	// Alarm_0403	403	Error	Wartość zadana wysokości jest większa od maksymalnej - zmień ustawienia w recepturze {0}
	//Error 7 - Bład nastaw max
	IF tonMaxHeightError.Q  THEN
		arfbAlarm[3].ipArguments.Clear() .AddLReal(lrMaxHeight);
		IF NOT arfbAlarm[3].bActive THEN
// 			bHeightMotorUp:=FALSE;
// 			bHeightMotorDown:=FALSE;
			arfbAlarm[3].Raise(nTimeStamp:=0);
		END_IF
	ELSE	
		IF  arfbAlarm[3].bActive AND bReset THEN
			arfbAlarm[3].Clear(nTimeStamp:=0, bResetConfirmation:= FALSE);
		END_IF	
// 		bError:=TRUE;
// 		udiErrorID:=7;
// 		udiErrorID:= udiErrorID+udiStationIndex;
// 		sErrorDescription:='Wartość zadana wysokości jest większa od maksymalnej - zmień ustawienia w recepturze';
// 		sErrorDescription2:=REAL_TO_STRING(LREAL_TO_INT(lrMaxHeight));
	END_IF
	// Alarm_0404	404	Error	Wartość zadana wysokości jest mniejsza od minimalnej - zmień ustawienia w recepturze {0}
	//Error 8 - Bład nastaw min
	IF tonMinHeightError.Q THEN
			arfbAlarm[4].ipArguments.Clear() .AddLReal(lrMinHeight);
		IF NOT arfbAlarm[4].bActive THEN
// 			bHeightMotorUp:=FALSE;
// 			bHeightMotorDown:=FALSE;
			arfbAlarm[4].Raise(nTimeStamp:=0);
		END_IF
	ELSE	
		IF  arfbAlarm[4].bActive AND bReset THEN
			arfbAlarm[4].Clear(nTimeStamp:=0, bResetConfirmation:= FALSE);
		END_IF
// 		bError:=TRUE;
// 		udiErrorID:=8;
// 		udiErrorID:= udiErrorID+udiStationIndex;
// 		sErrorDescription:='Wartość zadana wysokości jest mniejsza od minimalnej - zmień ustawienia w recepturze ';
// 		sErrorDescription2:=REAL_TO_STRING(LREAL_TO_INT(lrMinHeight));
	END_IF	
	// Alarm_0405	405	Error	Błąd falownika
	//Error 8 - Bład falownika
	IF tonInverterError.Q THEN
		IF NOT arfbAlarm[5].bActive THEN
			arfbAlarm[5].Raise(nTimeStamp:=0);
		END_IF
		IF arfbAlarm[5].bActive AND bReset THEN
			fbInverter.bReset := TRUE;
		END_IF
	ELSE	
		IF  arfbAlarm[5].bActive AND bReset THEN
			arfbAlarm[5].Clear(nTimeStamp:=0, bResetConfirmation:= FALSE);
		END_IF
// 		bError:=TRUE;
// 		udiErrorID:=9;
// 		udiErrorID:= udiErrorID+udiStationIndex;
// 		sErrorDescription:='Błąd falownika';
// 		sErrorDescription2:='';
	END_IF		
	
	
	
ELSE
	bError	:=FALSE;
END_IF


//-----------------------------------------------------------------------
IF bError AND NOT bStateError THEN

	IF eLastState = eRunning THEN
		bCycleNotDone						:= TRUE;
	END_IF

	eState 									:= E_Station.eError;
END_IF


//------------------------------------------------------------------------

(*Wyświetlanie błedu na wyjściu*)
bError							:= FALSE;
FOR nAlarmNumerator := 0 TO 19 DO
	bError						:= bError OR arfbAlarm[nAlarmNumerator].bActive;
END_FOR

(*Przepisywanie nazwy stacji*)
sErrorStationName 							:= WSTRING_TO_STRING(sStationName);

//Jezeli nie zbazowane to potrzebne bazowanie
IF NOT bHeightMotorEncoderHomed  THEN
	bHomingDone								:=	FALSE;
END_IF
END_ACTION

ACTION ACT_HeightMotor:
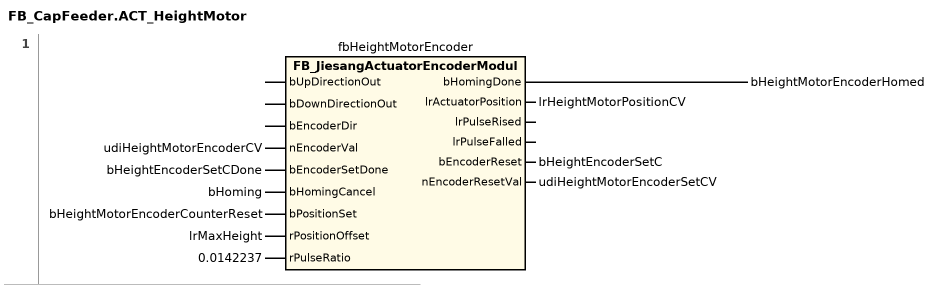
// NETWORK 1
fbHeightMotorEncoder(
    nEncoderVal := udiHeightMotorEncoderCV,
    bEncoderSetDone := bHeightEncoderSetCDone,
    bHomingCancel := bHoming,
    bPositionSet := bHeightMotorEncoderCounterReset,
    rPositionOffset := lrMaxHeight,
    rPulseRatio := 0.0142237,
    lrActuatorPosition => lrHeightMotorPositionCV,
    bEncoderReset => bHeightEncoderSetC,
    nEncoderResetVal => udiHeightMotorEncoderSetCV); // FB_JiesangActuatorEncoderModul
bHeightMotorEncoderHomed := fbHeightMotorEncoder.bHomingDone;
END_ACTION

ACTION ACT_Homing:
//BAZOWANIE

tofHeightMotorDown(IN:=bHeightMotorDown, PT:=T#1S); //Zabezpieczenie przed zbyt szybkim przełączeniem pomiędzy Down a Up, bezpiecznieki sie palą
	
//Podnoszenie stacji do maksymalnej pozycji
IF NOT bHeightMotorEncoderHomed OR rtEncoderHomed.Q THEN
	bHeightMotorUp:=(*TRUE*) NOT tofHeightMotorDown.Q AND NOT tonHomingSensor.Q;
	bHeightMotorDown:=FALSE;
	IF tonHeightNoChange.Q OR tonHeightNoChangeTime.Q THEN
		bHeightMotorEncoderCounterReset:=TRUE;
		bHeightMotorUp:=FALSE;
    END_IF
	//Jesli enkoder zbazowany zakończ bazowanie	
	IF rtEncoderHomed.Q  THEN
		bHeightMotorUp:=FALSE;
		bHeightMotorDown:=FALSE;
		eState:=E_Station.eHomingDone;
	END_IF		
		
//Po podniesieniu stacji opuszczanie do ustalonej wysokości
ELSIF bHeightMotorEncoderHomed THEN
	bHeightMotorEncoderCounterReset:=FALSE;
	bHeightMotorUp:=lrHeightMotorPositionCV<=lrHeightMotorPositionSV;
	bHeightMotorDown:=lrHeightMotorPositionCV>=lrHeightMotorPositionSV;
	//Kiedy stacja osiągnie wysokość zadaną
	IF ABS(lrHeightMotorPositionCV-lrHeightMotorPositionSV)<0.5 OR tonLimitPosMaxReachedDelay.Q OR tonLimitPosMinReachedDelay.Q THEN
		bHeightMotorDown:=FALSE;
		bHeightMotorUp:=FALSE;
		eState:=E_Station.eHomingDone;
	END_IF			
END_IF
END_ACTION

ACTION ACT_Inverter:
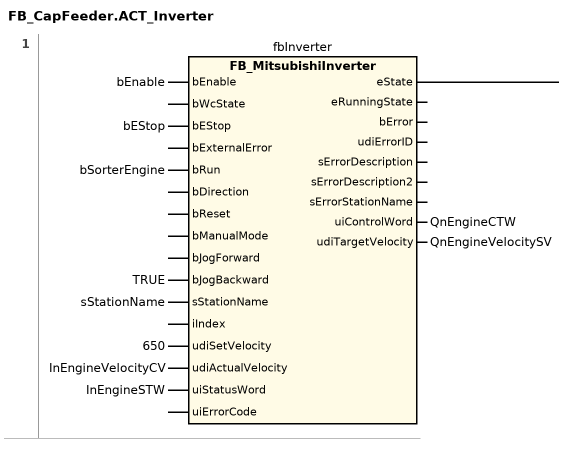
// NETWORK 1
fbInverter(
    bEnable := bEnable,
    bEStop := bEStop,
    bRun := bSorterEngine,
    bJogBackward := TRUE,
    sStationName := sStationName,
    udiSetVelocity := 650,
    udiActualVelocity := InEngineVelocityCV,
    uiStatusWord := InEngineSTW,
    uiControlWord => QnEngineCTW,
    udiTargetVelocity => QnEngineVelocitySV); // FB_MitsubishiInverter
END_ACTION

ACTION ACT_Limits:
IF iTimeToEmptySleeveError < 5 THEN
	iTimeToEmptySleeveError := 5;
END_IF
END_ACTION

ACTION ACT_ManualMovements:
//W trybie ruchów manualnych wykonuj ruchy za pomocą rozkazów manualnych
IF NOT bRun THEN
	
	bHeightMotorUp:=bManualHeightMotorUp;
	bHeightMotorDown:=bManualHeightMotorDown;
	bSorterEngine:=bManualSorterEngine;
	bSorterAir:=bManualSorterAir;
	
	bGate1:=bManualGate1; //Not dla tego, że defoltowy stan WYSUNIĘTY (true)
	bGate2:=bManualGate2; //Not dla tego, że defoltowy stan WYSUNIĘTY (true)

(*ELSE	//Kasuje zeby po cyklu nic sie nie poruszało

	bManualHeightMotorUp 	:= FALSE;
	bManualHeightMotorDown  := FALSE;
	bSorterEngine	:=FALSE;
	bSorterAir		:=FALSE;
*)	
END_IF


IF bHoming OR bHeightSet THEN
	eState:=E_Station.eHoming;
END_IF

IF bRun THEN	
	ACT_Running();
END_IF
//Zabezpieczenie przed kolizją stacji poprzez ruch podnośnika	
IF bHeightMotorDown AND lrHeightMotorPositionCV<=lrMinHeight AND NOT bHoming AND NOT bHeightSet THEN
	bHeightMotorDown:=FALSE;
END_IF	

IF bHeightMotorUp AND lrHeightMotorPositionCV>=lrMaxHeight AND NOT bHoming AND NOT bHeightSet THEN
	bHeightMotorUp:=FALSE;
END_IF
END_ACTION

ACTION ACT_ResetCommands:
//Reset komend ruchu 	


bHeightMotorUp				:=	FALSE;
bHeightMotorDown			:=	FALSE;
bSorterAir 		:= 	FALSE;
bSorterEngine 		:=	FALSE;
END_ACTION

ACTION ACT_Running:
//----------------------------------------------------------------------------------
// Obsługa podajnik zamknięc


(*CASE iValvesCycleCase OF
	0:
		bGate1:= FALSE;
		IF (tonGates1.Q) THEN
			iValvesCycleCase :=1;
		END_IF
	1:
		bGate1:= TRUE;
		IF (tonGates2.Q) THEN
			iValvesCycleCase :=2;
		END_IF	
	2:
		bGate2:= FALSE;
		IF (tonGates3.Q) THEN
			iValvesCycleCase :=3;
		END_IF
	3:
		bGate2:= TRUE;
		IF (tonGates4.Q) THEN
			iValvesCycleCase :=0;
		END_IF	
END_CASE*)

//rtOutSensor(CLK:=P08_CapSorter.IbCapSorterGateGateAfterSensor);
	
CASE iValvesCycleCase OF
	0:
		//IF (rtOutSensor.Q) THEN
		IF (NOT bSensorInPipe) THEN

			iValvesCycleCase:=1;
		END_IF
		;
	1:
		bGate1:= TRUE;
		IF (tonGates1.Q) THEN
			iValvesCycleCase :=2;
		END_IF
	2:
		bGate1:= FALSE;
		IF (tonGates2.Q) THEN
			iValvesCycleCase :=3;
		END_IF	
	3:
		bGate2:= TRUE;
		IF (tonGates3.Q) THEN
			iValvesCycleCase :=4;
		END_IF
	4:
		bGate2:= FALSE;
		IF (tonGates4.Q) THEN
			iValvesCycleCase :=0;
		END_IF	
END_CASE

CASE eRunningState OF
	
	//NIEGOTOWY
	E_CapFeederState.eDisabled:
		eRunningState:=E_CapFeederState.eReady;

	E_CapFeederState.eReady:
		iTryUnblockWheel		:=	0;
		bTryUnblockWheel		:= FALSE;	
		fbInverter.bDirection 	:= FALSE;
		IF bRun THEN
			eRunningState			:=E_CapFeederState.eSorting;
		END_IF
	
	
	E_CapFeederState.eSorting:
	
		bSorterEngine:=tonAirBeforeStart.Q;
		bSorterAir:=(	//Nie wiem co to za wymysły
						(aBufferedSensorValue[20](*tofCapFeederSorterCapSensor.Q*) OR NOT tonAirBeforeStart2.Q)(* AND bImpON*)AND NOT bBlowDelay
					)	OR	
					bTryUnblockWheel // Dmuchanie jeżeli jest obrót do tyłu
;
		//aBufferedSensorValue[20] - 20 to jest opóznenie (buferizacja signala czujnika w cyklach programy (3ms x 20 = 60 ms). Czas opóznenia 
		//możemy obliczyć od prędcosci falownika i prszykładni: mamy 51 gniazdk0, 800 rpm, przykladnia 1:40 => mamy 800/40=20rmp, /60 =>
		//0,33 obrota / sec => 0,33 obrota/sec * 51 dnazdko/obrot = 17 gniazdek/sek => 1/17 = 0,059sec/1gniazdko => opoznenie 60 ms
		//60ms/3ms(czas cyclu) => 20 cyclów
		
		(*Próba odblokowania koła*)
			iTryUnblockWheel := iTryUnblockWheel + 1;
			IF rtCapSorterSensor.Q THEN
				iTryUnblockWheel	:=	0;
			END_IF
			IF tonEngineBlocked.Q THEN
				bTryUnblockWheel := TRUE;
			END_IF	
			IF bTryUnblockWheel THEN
				fbInverter.bDirection := TRUE;
			END_IF
			IF tonTryUnblockWheel.Q THEN
				iTryUnblockWheel		:=	0;//dp
				bTryUnblockWheel		:= FALSE;
				fbInverter.bDirection 	:= FALSE;
			END_IF
		(* Koniec Próba odblokowania koła*)	
		
		IF tonSortingEngineOff.Q THEN 
			eRunningState 			:=E_CapFeederState.eSleeveFull;
		END_IF
	
	E_CapFeederState.eSleeveFull:
	
		bSorterEngine:=FALSE;
		bSorterAir:=NOT tonAirAfterStop.Q(* AND bImpON*);
		IF tonAirAfterStop.Q THEN
			IF tonSortingEngineOn.Q THEN
				eRunningState		:=E_CapFeederState.eSorting; 
			END_IF
		END_IF
	
	E_CapFeederState.eSleeveLowLevel:
	
			//Wlaczenie silnika i zaworu po czasie
		bSorterEngine:=TRUE;
		bSorterAir:=tofCapFeederSorterCapSensor.Q (*AND bImpON*);
		IF tonSortingEngineOff.Q THEN
			eRunningState		 	:=E_CapFeederState.eSorting;
		END_IF
	
END_CASE
END_ACTION

ACTION ACT_Signals:
(** Timery na potrzeby bazowania**)
rtEncoderHomed(CLK:=bHeightMotorEncoderHomed,Q=>);
tonHeightNoChange(IN:=((bHeightMotorUp OR bHeightMotorDown OR tonHomingSensor.Q) AND (lrLastHeightMotorPositionCV=lrHeightMotorPositionCV)), PT:=T#500MS); 
tonHomingSensor(IN:=(bHomingSensor), PT:=T#100MS);
//tonHeightNoChangeTime(IN:=(eState = E_Station.eHoming OR eState = E_Station.ePreparingToDisable) AND bHeightMotorUp, PT:=T#8S); 

tonLimitPosMinReachedDelay(IN:=(lrHeightMotorPositionCV<=lrMinHeight) AND eState=E_Station.eHoming,PT:=T#2S);
tonLimitPosMaxReachedDelay(IN:=(lrHeightMotorPositionCV>=lrMaxHeight) AND eState=E_Station.eHoming,PT:=T#2S);
	
(** Timery używane podczas pracy stacji**)
tonSortingEngineOff(IN:=((eRunningState=E_CapFeederState.eSorting OR eRunningState=E_CapFeederState.eSleeveLowLevel) AND bRun AND bFullSleeveSensor),PT:=INT_TO_TIME(iTimeDelayOff));
tonSortingEngineOn(IN:=((eRunningState=E_CapFeederState.eSorting OR eRunningState=E_CapFeederState.eSleeveFull) AND bRun AND NOT bFullSleeveSensor),PT:=INT_TO_TIME(iTimeDelayOn));
tonSleeveFullEngineOn(IN:=(eRunningState=E_CapFeederState.eSleeveFull AND bRun AND NOT bFullSleeveSensor),PT:=INT_TO_TIME(iTimeDelayOff));
rtCapSorterSensor(CLK:=bSorterCapSensor, Q=>);
tonEngineBlocked(IN:=iTryUnblockWheel > 1500 AND bSorterEngine AND NOT bTryUnblockWheel,PT:=T#1MS); //Zablokowany silnik
tonTryUnblockWheel(IN:=bTryUnblockWheel, PT:=T#1S900MS);
tofCapFeederSorterCapSensor(IN:=tonCapFeederSorterCapSensor.Q,PT:=T#100MS); //bylo 200
tonCapFeederSorterCapSensor(IN:=bSorterCapSensor,PT:=T#3mS);//było 3ms
tonAirBeforeStart(IN:=eRunningState=E_CapFeederState.eSorting, PT:=T#1S);
rtCapFeederSorterCapSensor(CLK:=tofCapFeederSorterCapSensor.Q,Q=>);

tonAirBeforeStart2(IN:=eRunningState=E_CapFeederState.eSorting, PT:=T#2S);
tonAirAfterStop(IN:=eRunningState=E_CapFeederState.eSleeveFull, PT:=T#2S);

//prszesunęcie wartosci czujnika po buforu opoznenia 

FOR i:=40 TO 1 BY -1 DO
	aBufferedSensorValue[i] := aBufferedSensorValue[i-1];
END_FOR
aBufferedSensorValue[0] := bSorterCapSensor;

IF rtCapFeederSorterCapSensor.Q THEN
	bBlowDelay := TRUE;
	
END_IF
tonbBlowDelay(IN:=bBlowDelay,PT:=T#35MS);
IF tonbBlowDelay.Q THEN
	bBlowDelay:= FALSE;
END_IF
TimerOn (IN := NOT bImpOn, PT := T#10MS);
IF TimerOn.Q THEN
	bImpOn := TRUE;
END_IF
TimerOff (IN := bImpOn, PT := T#10MS);
IF TimerOff.Q THEN
	bImpON := FALSE;
END_IF

//Czasówki pneumatiki
//tonGates1(IN:= (iValvesCycleCase = 0 AND (eState = E_Station.eRunning OR eState = E_Station.eManualMovement)), PT:=T#300MS);//150//300
//tonGates2(IN:= (iValvesCycleCase = 1 AND (eState = E_Station.eRunning OR eState = E_Station.eManualMovement)), PT:=T#200MS);//500//300
//tonGates3(IN:= (iValvesCycleCase = 2 AND (eState = E_Station.eRunning OR eState = E_Station.eManualMovement)), PT:=T#300MS);//150//300
//tonGates4(IN:= (iValvesCycleCase = 3 AND (eState = E_Station.eRunning OR eState = E_Station.eManualMovement)), PT:=T#200MS);//500//300

//Czasówki pneumatiki
tonGates1(IN:= (iValvesCycleCase = 1 AND (eState = E_Station.eRunning OR eState = E_Station.eManualMovement)), PT:=T#200MS);//150//300
tonGates2(IN:= (iValvesCycleCase = 2 AND (eState = E_Station.eRunning OR eState = E_Station.eManualMovement)), PT:=T#200MS);//500//300
tonGates3(IN:= (iValvesCycleCase = 3 AND (eState = E_Station.eRunning OR eState = E_Station.eManualMovement)), PT:=T#200MS);//150//300
tonGates4(IN:= (iValvesCycleCase = 4 AND (eState = E_Station.eRunning OR eState = E_Station.eManualMovement)), PT:=T#200MS);//500//300


(** Dodatkowy timer przy zatrzymywaniu**)
tonStoppingTime( IN:= eState= E_Station.eStopping, PT:=T#2S);
END_ACTION

ACTION ACT_Statistic:
//Statystyka do zliczania czasu cyklu 
rtrigCycleTimerRead(CLK:=eRunningState=E_CapFeederState.eSleeveFull OR eRunningState=E_CapFeederState.eSleeveLowLevel);

	IF rtrigCycleTimerRead.Q THEN
		tCycleTime:=tonCycleTimer.ET;
		
	END_IF
	
tonCycleTimer(IN:=eRunningState= E_CapFeederState.eSorting , PT:=T#1D);
END_ACTION

ACTION ACT_Status:

(*Zapisywanie ostatniego stanu*)
	IF eLastStateTemp<>eState THEN
		eLastState := eLastStateTemp;
	END_IF
	eLastStateTemp := eState;
	
	IF eLastRunningStateTemp<>eRunningState THEN
		eLastRunningState := eLastRunningStateTemp;
	END_IF
	eLastRunningStateTemp := eRunningState;
(*Koniec Zapisywanie ostatniego stanu*)
END_ACTION

ACTION ACT_Warnings:
//Usrawianie warningów

//Filtrowanie czujnika ultradźwiękowego
fbbLevelSensor	(bIN:=NOT bLevelSensor AND (eRunningState=E_CapFeederState.eSorting OR eRunningState=E_CapFeederState.eSleeveLowLevel OR eRunningState=E_CapFeederState.eSleeveFull) , tFilterTimeOn:= T#5S, tFilterTimeOff:=T#5S , bOUT=> );


IF fbbLevelSensor.bOUT THEN
		bWarning1						:=	TRUE;			
		udiWarningID					:=	1;
		sWarningDescription				:=	'Nieski poziom w sorterze nasadek';
ELSE
		bWarning1						:=	FALSE;			
		udiWarningID					:=	0;
		sWarningDescription				:=	'';
END_IF
END_ACTION

ACTION aStationID:
udiStationID	:=	iStationIndex;
END_ACTION

END_FUNCTION_BLOCK

// ---- POUs/P01_BottleFeeder.TcPOU
(*
Nazwa:			P01_BottleFeeder
Opis:			Stacja podajnika nasadek
Wersja:			v0.1
Data:			2018-10-10
Autor:			DP
Urzadzenia:		
Konfiguracja:	
Info:

*)
PROGRAM P01_BottleFeeder
VAR_INPUT
	IbBottleFeederGate1Sensor					:BOOL;			// Czujnik otwarcia 1 szlabanu 
	IbBottleFeederGate2Sensor					:BOOL;			// Czujnik otwarcia 2 szlabanu 
	IbBottleFeederArmLeftSensor					:BOOL;			// Czujnik położenia siłownika poziomego ramienia - lewy
	IbBottleFeederArmRightSensor				:BOOL;			// Czujnik położenia siłownika poziomego ramienia - prawy
	IbBottleFeederArmUpSensor					:BOOL;			// Czujnik położenia siłownika pionowego ramienia - góra
	IbBottleFeederArmDownSensor					:BOOL;			// Czujnik polożenia siłowniak pionowego ramienia - dół
	IbBottleFeederFormPositioningClosedSensor	:BOOL;			// Czujnik schowania siłownika pozycjonujacego formatke
	IbBottleFeederBottleSensor					:BOOL;			// Czujnik obecności butelki pomiedzy szlabanami
	IbBottleFeederFormGateBeforeSensor 			:BOOL;			// Czujnik przed szlabanem formatek
	IbBottleFeederFormGateAfterSensor 			:BOOL;			// Czujnik za szlabanem formatek
	IbBottleFeederLevelSensor					:BOOL;			// Czujnik kolejki butelki
	IbBottleFeederNotInsertedSensor				AT %I*: BOOL; 	// Czujnik źle włozonej butelki za stacją	
	
END_VAR

VAR
	tonSimu1	:	TON;
	tonSimu2	:	TON;	
	tonSimu3	:	TON;	

	fbBottleFeeder						  	: FB_BottleFeeder;		// Bloczek do obsługi stacji podajnika butelek
	fbTurnTable								: FB_MitsubishiInverter; 	//Bloczek do obsługi falownika stołu obrotewego
	
	eBottleFeederStationState				: E_Station;
	eBottleFeederRunningState				: E_BottleFeederState;
	fbBottleFeederState						: FB_State;
	
	eBottleFeederTurnTableState				: E_Station;
	eBottleFeederTurnTableRunningState		: E_ConveyorState;
	fbBottleSorterTurnTableState			: FB_State;
	
	fbGateBottleFeeder						: FB_SpringGateV2;
	
	//Wyjścia sterujące
	QbBottleFeederGate1						:BOOL;			// Szlaban 1 (lewy)
	QbBottleFeederGate2						:BOOL;			// Szlaban 2 (prawy)
	QbBottleFeederArmLeft					:BOOL;			// Lewo
	QbBottleFeederArmDown					:BOOL;			// Dół
	QbBottleFeederGripper					:BOOL;			// Chwytak
	QbBottleFeederFormPositioning			:BOOL;			// Pozycjonowanie formatki
	QbBottleFeederFormGate					:BOOL;			// Szlaban formatki
	
	// Stół obrotowy
	uiBottleFeederTurnTableSW					AT %I*: UINT;
	uiBottleFeederTurnTableActualVelocity		AT %I*: UDINT;
	uiBottleFeederTurnTableCW  					AT %Q*: UINT;
	udiBottleFeederTurnTableVelocity			AT %Q*: UDINT;
	bGateRun: BOOL;
	iTest2: INT;
	bTestTurnTableRun: BOOL;
	
	bTest: BOOL;
	tonNotQbBottleFeederArmDown: TON;
END_VAR

aWarning();
aBottleFeeder();
aTurntable();
aGateTime();
aGate();

tonNotQbBottleFeederArmDown(IN:= NOT QbBottleFeederArmDown, PT:=T#50MS);


VIS.nBottleFeederTurnTableVelocityCV := uiBottleFeederTurnTableActualVelocity;

IF fbBottleFeeder.bCycleDone THEN
	bGateRun:=TRUE;
END_IF

IF fbGateBottleFeeder.bCycleDone THEN
	bGateRun:=FALSE;
END_IF

(********ASOWANIE ROZKAZÓW CYKLI*********)
IF fbBottleFeeder.bCycleDone AND bManualMode THEN
	VIS.bBottleFeederRun := FALSE;
END_IF


fbBottleFeederState(
	eState									:= eBottleFeederStationState,
	bRun									:= VIS.bBottleFeederRun,
	eBottleSorterRunningState				:= eBottleFeederRunningState,
	sStateDesc								=> VIS.sBottleFeederState,
	iState									=> VIS.iBottleFeederState);
	
(*
// tutaj dorobić obsługe wizki dla stoli obrotowego
eBottleSorterTurnTableRunningState:=eBottleSorterTurnTableState;


fbBottleSorterTurnTableState(
	eState													:= eBottleSorterTurnTableState , 
	bRun													:= GVL.bBottleSorterTurnTableRun,	
	eBottleSorterRunningState									:= eBottleSorterTurnTableRunningState , 
	sStateDesc												=> VIS.sBottleSorterTurnTableState,
	iState													=> VIS.iBottleSorterTurnTableState	);
*)

ACTION aBottleFeeder:
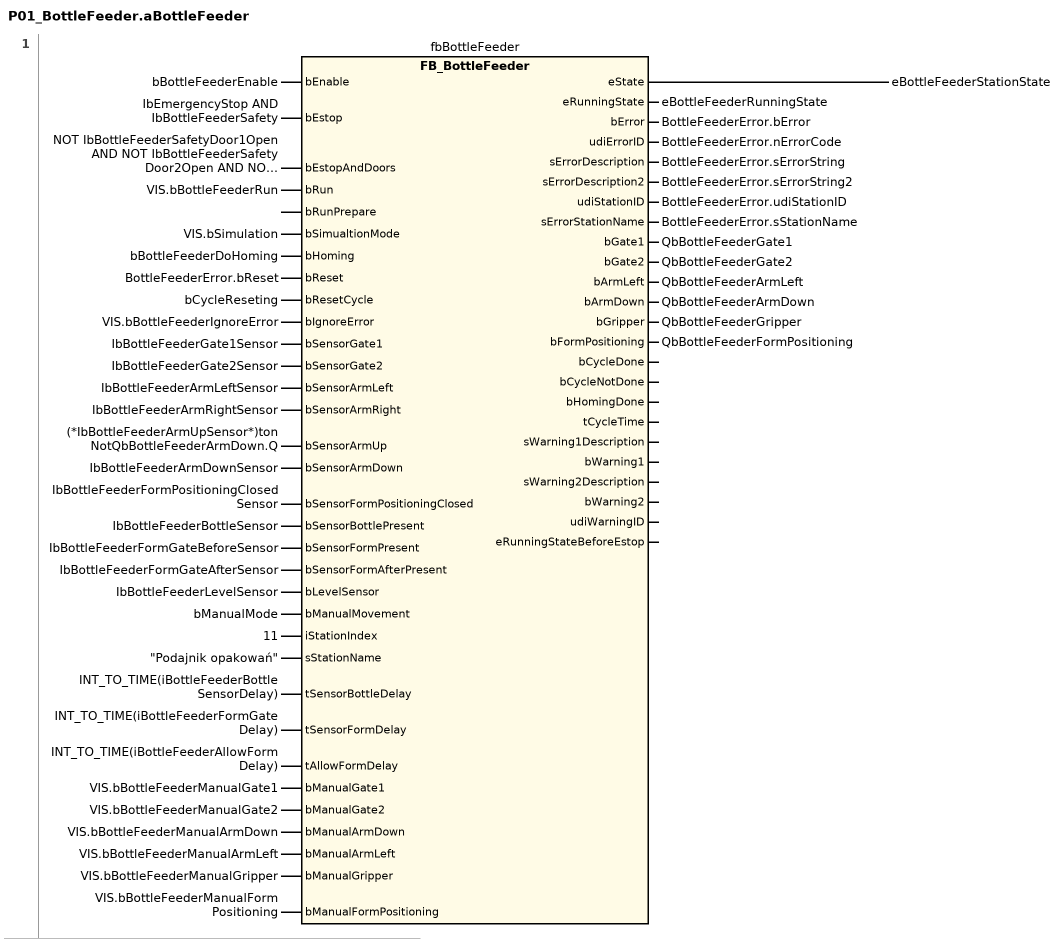
// NETWORK 1
fbBottleFeeder(
    bEnable := bBottleFeederEnable,
    bEstop := IbEmergencyStop AND IbBottleFeederSafety,
    bEstopAndDoors := NOT IbBottleFeederSafetyDoor1Open AND NOT IbBottleFeederSafetyDoor2Open AND NOT IbBottleFeederSafetyDoor3Open,
    bRun := VIS.bBottleFeederRun,
    bSimualtionMode := VIS.bSimulation,
    bHoming := bBottleFeederDoHoming,
    bReset := BottleFeederError.bReset,
    bResetCycle := bCycleReseting,
    bIgnoreError := VIS.bBottleFeederIgnoreError,
    bSensorGate1 := IbBottleFeederGate1Sensor,
    bSensorGate2 := IbBottleFeederGate2Sensor,
    bSensorArmLeft := IbBottleFeederArmLeftSensor,
    bSensorArmRight := IbBottleFeederArmRightSensor,
    bSensorArmUp := (*IbBottleFeederArmUpSensor*)tonNotQbBottleFeederArmDown.Q,
    bSensorArmDown := IbBottleFeederArmDownSensor,
    bSensorFormPositioningClosed := IbBottleFeederFormPositioningClosedSensor,
    bSensorBottlePresent := IbBottleFeederBottleSensor,
    bSensorFormPresent := IbBottleFeederFormGateBeforeSensor,
    bSensorFormAfterPresent := IbBottleFeederFormGateAfterSensor,
    bLevelSensor := IbBottleFeederLevelSensor,
    bManualMovement := bManualMode,
    iStationIndex := 11,
    sStationName := "Podajnik opakowań",
    tSensorBottleDelay := INT_TO_TIME(iBottleFeederBottleSensorDelay),
    tSensorFormDelay := INT_TO_TIME(iBottleFeederFormGateDelay),
    tAllowFormDelay := INT_TO_TIME(iBottleFeederAllowFormDelay),
    bManualGate1 := VIS.bBottleFeederManualGate1,
    bManualGate2 := VIS.bBottleFeederManualGate2,
    bManualArmDown := VIS.bBottleFeederManualArmDown,
    bManualArmLeft := VIS.bBottleFeederManualArmLeft,
    bManualGripper := VIS.bBottleFeederManualGripper,
    bManualFormPositioning := VIS.bBottleFeederManualFormPositioning,
    eRunningState => eBottleFeederRunningState,
    bError => BottleFeederError.bError,
    udiErrorID => BottleFeederError.nErrorCode,
    sErrorDescription => BottleFeederError.sErrorString,
    sErrorDescription2 => BottleFeederError.sErrorString2,
    udiStationID => BottleFeederError.udiStationID,
    sErrorStationName => BottleFeederError.sStationName,
    bGate1 => QbBottleFeederGate1,
    bGate2 => QbBottleFeederGate2,
    bArmLeft => QbBottleFeederArmLeft,
    bArmDown => QbBottleFeederArmDown,
    bGripper => QbBottleFeederGripper,
    bFormPositioning => QbBottleFeederFormPositioning); // FB_BottleFeeder
eBottleFeederStationState := fbBottleFeeder.eState;
END_ACTION

ACTION aGate:
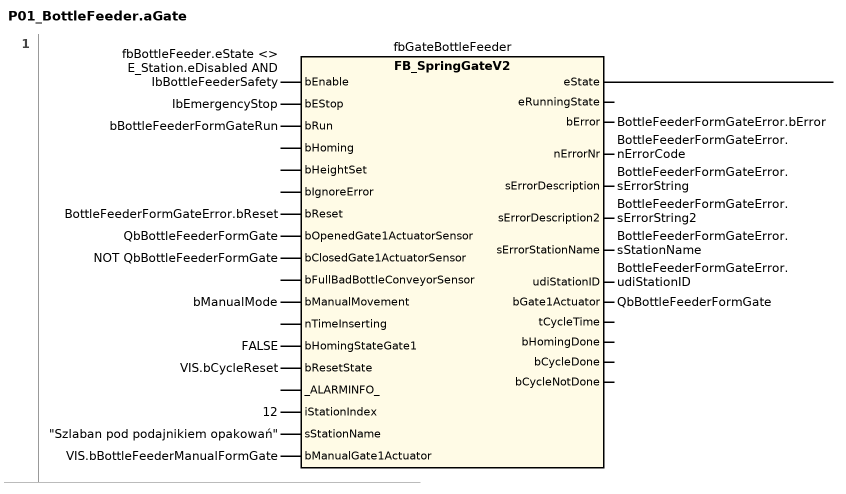
// NETWORK 1
fbGateBottleFeeder(
    bEnable := fbBottleFeeder.eState <> E_Station.eDisabled AND IbBottleFeederSafety,
    bEStop := IbEmergencyStop,
    bRun := bBottleFeederFormGateRun,
    bReset := BottleFeederFormGateError.bReset,
    bOpenedGate1ActuatorSensor := QbBottleFeederFormGate,
    bClosedGate1ActuatorSensor := NOT QbBottleFeederFormGate,
    bManualMovement := bManualMode,
    bHomingStateGate1 := FALSE,
    bResetState := VIS.bCycleReset,
    iStationIndex := 12,
    sStationName := "Szlaban pod podajnikiem opakowań",
    bManualGate1Actuator := VIS.bBottleFeederManualFormGate,
    bError => BottleFeederFormGateError.bError,
    nErrorNr => BottleFeederFormGateError.nErrorCode,
    sErrorDescription => BottleFeederFormGateError.sErrorString,
    sErrorDescription2 => BottleFeederFormGateError.sErrorString2,
    sErrorStationName => BottleFeederFormGateError.sStationName,
    udiStationID => BottleFeederFormGateError.udiStationID,
    bGate1Actuator => QbBottleFeederFormGate); // FB_SpringGateV2
END_ACTION

ACTION aGateTime:
IF bFormTransportersDispencerSlowSpeed THEN 
	fbGateBottleFeeder.nTimeInserting	:=	500;
ELSE
	fbGateBottleFeeder.nTimeInserting	:=	200;	//200
END_IF
END_ACTION

ACTION aTurntable:
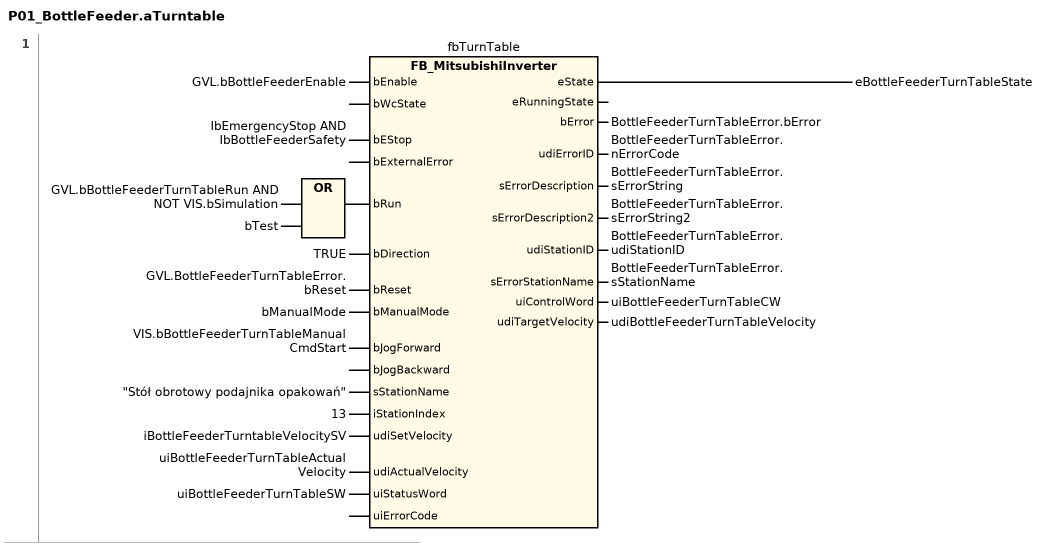
// NETWORK 1
fbTurnTable(
    bEnable := GVL.bBottleFeederEnable,
    bEStop := IbEmergencyStop AND IbBottleFeederSafety,
    bRun := (GVL.bBottleFeederTurnTableRun AND NOT VIS.bSimulation) OR bTest,
    bDirection := TRUE,
    bReset := GVL.BottleFeederTurnTableError.bReset,
    bManualMode := bManualMode,
    bJogForward := VIS.bBottleFeederTurnTableManualCmdStart,
    sStationName := "Stół obrotowy podajnika opakowań",
    iStationIndex := 13,
    udiSetVelocity := iBottleFeederTurntableVelocitySV,
    udiActualVelocity := uiBottleFeederTurnTableActualVelocity,
    uiStatusWord := uiBottleFeederTurnTableSW,
    bError => BottleFeederTurnTableError.bError,
    udiErrorID => BottleFeederTurnTableError.nErrorCode,
    sErrorDescription => BottleFeederTurnTableError.sErrorString,
    sErrorDescription2 => BottleFeederTurnTableError.sErrorString2,
    udiStationID => BottleFeederTurnTableError.udiStationID,
    sErrorStationName => BottleFeederTurnTableError.sStationName,
    uiControlWord => uiBottleFeederTurnTableCW,
    udiTargetVelocity => udiBottleFeederTurnTableVelocity); // FB_MitsubishiInverter
eBottleFeederTurnTableState := fbTurnTable.eState;
END_ACTION

ACTION aWarning:
// Warning 1
IF (IbBottleFeederSafetyDoor3Open AND bBottleFeederEnable) AND NOT BottleFeederWarning[0].bWarning THEN
	BottleFeederWarning[0].bWarning										:=TRUE;
	BottleFeederWarning[0].udiWarningCode								:=1;
	BottleFeederWarning[0].sDescription									:='Podajnik butelek | Otwarte drzwi dostępowe';
ELSIF (NOT GVL_io.IbBottleFeederSafetyDoor3Open OR NOT bBottleFeederEnable) (*AND BottleFeederWarning[0].bAcknowledge*) THEN
	BottleFeederWarning[0].bWarning										:= FALSE;
	BottleFeederWarning[0].bAcknowledge									:= FALSE;
	VIS.uliWarningAcknowledge.23 										:= FALSE;
//ELSIF BottleFeederWarning[0].bAcknowledge THEN
//ELSE
//	BottleFeederWarning[0].bAcknowledge									:= TRUE;
END_IF	

(*// Warning 2
IF (fbBottleFeeder.bWarning1 AND bBottleFeederEnable) AND NOT BottleFeederWarning[1].bWarning THEN
	BottleFeederWarning[1].bWarning										:= TRUE;
	BottleFeederWarning[1].udiWarningCode								:= 2;
	BottleFeederWarning[1].sDescription									:= 'Podajnik butelek | Niski poziom butelek';
ELSIF (NOT fbBottleFeeder.bWarning1 OR NOT bBottleFeederEnable) AND BottleFeederWarning[1].bAcknowledge THEN
	BottleFeederWarning[1].bWarning										:= FALSE;
	BottleFeederWarning[1].bAcknowledge									:= FALSE;
	VIS.uliWarningAcknowledge.26 										:= FALSE;
ELSIF BottleFeederWarning[1].bAcknowledge THEN
	BottleFeederWarning[1].bAcknowledge									:= TRUE;
END_IF*)

//Warning 3
IF (IbBottleFeederSafetyDoor1Open AND bBottleFeederEnable) AND NOT BottleFeederWarning[2].bWarning THEN
	BottleFeederWarning[2].bWarning										:=TRUE;
	BottleFeederWarning[2].udiWarningCode								:=3;
	BottleFeederWarning[2].sDescription									:='Podajnik butelek | Otwarta bramka wjazdowa';
ELSIF (NOT IbBottleFeederSafetyDoor1Open OR NOT bBottleFeederEnable) (*AND BottleFeederWarning[2].bAcknowledge*) THEN
	BottleFeederWarning[2].bWarning										:= FALSE;
	BottleFeederWarning[2].bAcknowledge									:= FALSE;
	VIS.uliWarningAcknowledge.41 										:= FALSE;
//ELSIF BottleFeederWarning[2].bAcknowledge THEN
//	BottleFeederWarning[2].bAcknowledge									:= TRUE;
END_IF	

//Warning 4
BottleFeederWarning[3].sDescription										:='Podajnik butelek | Otwarta bramka wyjazdowa';
IF (IbBottleFeederSafetyDoor2Open AND bBottleFeederEnable) AND NOT BottleFeederWarning[3].bWarning THEN
	BottleFeederWarning[3].bWarning										:=TRUE;
	BottleFeederWarning[3].udiWarningCode								:=4;
	BottleFeederWarning[3].sDescription									:='Podajnik butelek | Otwarta bramka wyjazdowa';
ELSIF (NOT GVL_io.IbBottleFeederSafetyDoor2Open OR NOT bBottleFeederEnable) (*AND BottleFeederWarning[3].bAcknowledge*) THEN
	BottleFeederWarning[3].bWarning										:= FALSE;
	BottleFeederWarning[3].bAcknowledge									:= FALSE;
	VIS.uliWarningAcknowledge.42 										:= FALSE;
//ELSIF BottleFeederWarning[3].bAcknowledge THEN
//	BottleFeederWarning[3].bAcknowledge									:= TRUE;
END_IF
END_ACTION

END_PROGRAM

// ---- POUs/FB/NewFBs/FB_BottleFeeder.TcPOU
(*
Nazwa:	FB_BottleSorter
Opis:	Podajnik opakowań do formatek
Wersja:	V0.4
Data:	10.12.2024
Autor:	DP
Urządzenia:	Szlabany docisku opakowań, pneumatyczne podnoszenie opakowań, szlabany formatki
Konfiguracja:	
Info:
Zmiany:
- [12.12.2024] CycleReset, LastStaty
- [31.10.2024] DP na nowo
- [11.07.2023] DP dodano opcję wypuszczania pustych formatek po czasie (zyczenie anglikow)

*)

FUNCTION_BLOCK FB_BottleFeeder
VAR_INPUT
	bEnable						: BOOL;					// Załączenie stacji 
	bEstop						: BOOL;					// Stop awaryjny
	bEstopAndDoors				: BOOL;					// Drzwi zamknięte	
	bRun						: BOOL;					// Rozkaz pracy
	bRunPrepare					: BOOL;					// Przygotowanie do rozpoczecia pracy
	bSimualtionMode				: BOOL;					// Bit od symulacji czujnika butelki 
	bHoming						: BOOL;					// Bazowanie stacji 
	bReset						: BOOL;					// Resetowanie błędów stacji
	bResetCycle					: BOOL;					// Reset cyklu 
	bIgnoreError				: BOOL;					// Ignorowanie błędów
	bSensorGate1				: BOOL;					// Czujnik siłownika szlabanu 1 / wsunięty
	bSensorGate2				: BOOL;					// Czujnik siłownika szlabanu 2 / wsunięty
	bSensorArmLeft				: BOOL;					// Czujnik siłownika poziomiego / wsunięty
	bSensorArmRight				: BOOL;					// Czujnik siłownika poziomego	/ wysunięty
	bSensorArmUp				: BOOL;					// Czujnik siłownika pionowego / wsunięty
	bSensorArmDown				: BOOL;					// Czujnik siłowniak pionowego / wysunięty
	bSensorFormPositioningClosed: BOOL;					// Czujnik pozycjonowania formatek schowany
	bSensorBottlePresent		: BOOL;					// Czujnik obecności opakowania 
	bSensorFormPresent			: BOOL;					// Czujnik obecności formatki
	bSensorFormAfterPresent		: BOOL;					// Czujnik braku obecności formatki za podajnikiem
	bLevelSensor				: BOOL;					// Czujnik poziomu
	bManualMovement				: BOOL;					// Zezwolenie na ręczne ruchy 	
	iStationIndex				: UDINT;				// Indywidualny numer stacji
	sStationName				: WSTRING;				// Nazwa stacji

	tSensorBottleDelay			: TIME;					// Czasówka na dojazd butelki do czujnika na bramkach wjazdowyuch
	tSensorFormDelay			: TIME;					// Czasówka na stabilizacje formatki pod podajnikiem
	tAllowFormDelay				: TIME;
END_VAR

VAR_OUTPUT
	                     
	eState						: E_Station;
	eRunningState				: E_BottleFeederState;	// Stan przeciągania formatek
	bError						: BOOL;					// Błąd stacji
	udiErrorID					: UDINT;				// Nr blędu przeciągania formatek
	sErrorDescription			: STRING(200);			// Opis błędu
	sErrorDescription2			: STRING(200);			// Opis błędu
	udiStationID				: UDINT;				// Nr stacji	
	sErrorStationName			: STRING;				// Nazwa stacji
	bGate1						: BOOL;					// Otwarcie szlabanu 1 / wysnięty (opakowania)							
	bGate2						: BOOL;					// Otwarcie szlabanu 2 / wysnięty (opakowania)				
	bArmLeft					: BOOL;					// Lewo
	bArmDown					: BOOL;					// Dół
	bGripper					: BOOL;					// Chwytak
	bFormPositioning			: BOOL;					// Pozycjonowanie formatek

	bCycleDone					: BOOL;					// Sygnał zakończenia cyklu
	bCycleNotDone				: BOOL;					// Sygnał błędnego zakończenia cyklu 
	bHomingDone					: BOOL;					// Sygnał zbazowania stacji 
	tCycleTime					: TIME;					// Czas syklu stacji 
	sWarning1Description		: STRING;
	bWarning1					: BOOL;
	sWarning2Description		: STRING;
	bWarning2					: BOOL;
	udiWarningID				: UDINT;	
	
	eRunningStateBeforeEstop	: E_BottleFeederState; 	// Stan przed Estope
	
END_VAR

VAR_IN_OUT
	
	bManualGate1				: BOOL;					// Szlaban 1 - lewy
	bManualGate2				: BOOL;					// Szlaban 2 - lewy
	bManualArmDown				: BOOL;					// W dół
	bManualArmLeft				: BOOL;					// Lewo
	bManualGripper				: BOOL;					// Chwytak
	bManualFormPositioning		: BOOL;					// Pozycjonowanie formatki


END_VAR

VAR
	// State
	eLastState									: E_Station;						//Stan ogólny bloku
	eLastStateTemp								: E_Station;						//Stan ogólny bloku
	eLastRunningState							: E_BottleFeederState;				//Stan podbloku
	eLastRunningStateTemp						: E_BottleFeederState;				//Stan podbloku
	
	//Reset 
	rtResetCycle: R_TRIG;			
	rtrigCycleTimerRead							: R_TRIG;							// Do zliczania czasu
	tonCycleTimer								: TON;								// Timer

	//Triggery
	ftIbSensorLifterDown						: F_TRIG;							// Triger zjazdu z dolnego czujnika
	
	// czasówki
	tonPreparingToDisabled						: TON;								// Czasówka za długiego przygotowania do gotowosic
	tonPreparingToReadyOn						: TON;								// Czasówka za długiego przygotowania do gotowosic
	tonBottleSensorDelay						: TON;								// Czasówka na załączenie wykrycia butelki
	tonAllowEmptyForm							: TON;
	tonFormsPresentDelay						: TON;								// Czasówka na załączenie obecności formatki
	
	//czasówki od błędów	
	tonGate1Error								: TON;				
	tonGate2Error								: TON;
	tonArmLeftPositionError						: TON;
	tonArmRightPostionError						: TON;
	tonArmUpPositionError						: TON;
	tonArmDownPositionError						: TON;
	tonBottleAndFormTooLong						: TON;
	
	// case
	iHomingStep									: INT;
	
	// bit bledow
	bStateError									: BOOL;
	
	//Warning
	fbLevelSensor								:FB_InputFilter_v2;

	bSimulationSensor							: BOOL;
	tonEstopDelay: TON;
	bGate1LastState : BOOL;			
	bGate2LastState : BOOL;				
	bArmDownLastState : BOOL;				
	bArmLeftLastState : BOOL;				
	bGripperLastState : BOOL;				
	bFormPositioningLastState : BOOL;	
	tonGripper: TON;
	tonOpenedGripper: TON;
	tofRunning: TOF;
	tonArmDown: TON;
	
	//Zmienne od EVENTLOGGER
	bAlarmInit 						: BOOL := TRUE; 
	nAlarmNumerator					: INT;
	arfbAlarm						: ARRAY[0..19] OF  FB_TcAlarm;		//Tablica bloczków błędów
	fbSourceInfo 					: FB_TcSourceInfo;
	iSourceInfo						: I_TcSourceInfo;
	sAlarmTest						: STRING;
	//Koniec zmiennych od EVENTLOGGER
END_VAR

aLimits();
aErrorHandling();
aSignals();
aControl();
aStatistic();
aWarnings();
aStationID();
aCycleReset();
(*Zapisywanie ostatniego stanu*)
IF eLastStateTemp<>eState THEN
	eLastState := eLastStateTemp;
END_IF
eLastStateTemp := eState;
IF eLastRunningStateTemp<>eRunningState THEN
	eLastRunningState := eLastRunningStateTemp;
END_IF
eLastRunningStateTemp := eRunningState;
(*Koniec Zapisywanie ostatniego stanu*)

ACTION aControl:

//Wyłączenie stacji
IF NOT bEnable THEN
	IF eState <> E_Station.eRunning AND eState <> E_Station.eDisabled AND eState <> E_Station.ePreparingToDisable THEN
		eState										:=	E_Station.ePreparingToDisable;
	END_IF
END_IF
	
// Praca po Estopie
IF NOT bEstop  THEN	
	IF eState <> E_Station.eAborted AND eState <> E_Station.eAborting AND eState <> E_Station.eDisabled THEN
			eRunningStateBeforeEStop				:=	eRunningState;
			eState 									:=	E_Station.eAborting; 
	END_IF
END_IF
	
CASE eState OF
//--------------------------------------------------------------------------------
	E_Station.eDisabled:
		IF bEnable THEN
			eState									:=	E_Station.ePreparingToReady;
		END_IF
	
//-------------------------------------------------------------------------------
	E_Station.ePreparingToDisable:
		bGripper 									:= FALSE;
		bGate1										:= FALSE;	
		bGate2										:= TRUE;
		bArmDown									:= FALSE;
		bArmLeft									:= FALSE;
		bFormPositioning							:= FALSE;

		IF  tonPreparingToDisabled.Q THEN
			eState									:= E_Station.eDisabled;
			eRunningState							:= E_BottleFeederState.eDisabled;
		END_IF

//--------------------------------------------------------------------------------
	E_Station.eAborted:
		IF bEstop THEN
			eState									:= E_Station.ePreparingToReady;
		END_IF

//--------------------------------------------------------------------------------	
	E_Station.eAborting:
		aResetCommands();
		eState										:= E_Station.eAborted;
		eRunningState								:= E_BottleFeederState.eDisabled;

//--------------------------------------------------------------------------------
	E_Station.eError:
		IF bReset THEN
			eState									:= E_Station.eResetting;
			bError									:= FALSE;
		END_IF

//--------------------------------------------------------------------------------
	E_Station.eResetting:
		IF NOT bError THEN
			udiErrorID								:= 0;
			sErrorDescription						:= '';
			sErrorDescription2						:= '';
			eState									:= E_Station.ePreparingToReady;
		END_IF

//--------------------------------------------------------------------------------			
	E_Station.eManualMovement: 
		aManualMovements();
		IF NOT bManualMovement THEN
			bGate1									:=	bGate1LastState;			
			bGate2			    					:=  bGate2LastState;			
			bArmLeft		    					:=  bArmLeftLastState;		
			bArmDown		    					:=  bArmDownLastState;		
			bGripper		    					:=  bGripperLastState;		
			bFormPositioning    					:=  bFormPositioningLastState;
			eState									:=	E_Station.eReady;
		END_IF
		
//--------------------------------------------------------------------------------
	E_Station.eHoming: 			
		bHomingDone 								:= FALSE;
		aHoming();
		IF NOT bHoming	THEN
			eState									:= E_Station.ePreparingToReady;
		END_IF

//--------------------------------------------------------------------------------	
	E_Station.eHomingDone:
		bHomingDone									:= TRUE;
		IF NOT bHoming	THEN
			eState									:= E_Station.ePreparingToReady;
		END_IF

//--------------------------------------------------------------------------------				
	E_Station.ePreparingToReady:

		bGate1										:= FALSE;
		bGate2										:= TRUE;			
		bArmLeft									:= FALSE;
		bArmDown									:= FALSE;	
		bGripper									:= FALSE;
		bFormPositioning							:= FALSE;
	
		IF tonPreparingtoReadyOn.Q THEN
			eState									:= E_Station.eReady;
			eRunningState							:= E_BottleFeederState.eReady;
		END_IF

//--------------------------------------------------------------------------------
// Stan gotowości
		
	E_Station.eReady:
		
		IF bRunPrepare OR bRun AND (NOT bCycleDone AND NOT bCycleNotDone) THEN
			eState									:= E_Station.eStarting;
		END_IF
		
		IF bHoming THEN
			eState									:= E_Station.eHoming;
		END_IF
		
		IF bManualMovement THEN
			bManualGate1							:=	bGate1LastState				:= bGate1;			
			bManualGate2							:=  bGate2LastState			    := bGate2;			
			bManualArmDown							:=  bArmDownLastState			:= bArmDown;				
			bManualArmLeft							:=  bArmLeftLastState			:= bArmLeft;			
			bManualGripper							:=  bGripperLastState			:= bGripper;				
			bManualFormPositioning					:=  bFormPositioningLastState	:= bFormPositioning;	
			eState									:=	E_Station.eManualMovement;
			eRunningState							:=	E_BottleFeederState.eReady;
		END_IF
		
		IF NOT bRun  THEN
			bCycleDone								:=	FALSE;
			bCycleNotDone 							:=	FALSE;
		END_IF

//--------------------------------------------------------------------------------
	E_Station.eStopping:
	
		aRunning();
		IF eRunningState =	E_BottleFeederState.eReady OR eRunningState	= E_BottleFeederState.ePreparingToMove THEN
			eRunningState							:=	E_BottleFeederState.eReady;
			eState									:=	E_Station.eReady;
		END_IF
		IF eRunningState =	E_BottleFeederState.eGoAbove THEN
			eState									:=	E_Station.eReady;
		END_IF
		
//--------------------------------------------------------------------------------
	E_Station.eStarting:
	
		eState										:=	E_Station.eRunning;

//--------------------------------------------------------------------------------
	E_Station.eRunning:	
		
		aRunning();
		IF NOT bRun	THEN
			eState									:=	E_Station.eStopping;
		END_IF

		IF bCycleDone OR bCycleNotDone THEN (*Cykl zakończony*)
			eState									:=	E_Station.eReady;
		END_IF
		
END_CASE
END_ACTION

ACTION aCycleReset:
IF bResetCycle THEN
	aHoming();																
END_IF
END_ACTION

ACTION aErrorHandling:
// Alarm_0140	140	Error	Blokada otwarcia siłownika wjazdu opakowania - lewy - popraw lub usuń opakowanie
// Alarm_0141	141	Error	Blokada otwarcia siłownika wjazdu opakowania - prawy - popraw lub usuń opakowanie
// Alarm_0142	142	Error	Blokada lewej pozycji siłownika chwytaka - sprawdź położenie ramienia
// Alarm_0143	143	Error	Blokada prawej pozycji siłownika chwytaka - sprawdź położenie ramienia
// Alarm_0144	144	Error	Blokada górnej pozycji siłownika chwytaka - sprawdź położenie ramienia lub usuń opakowanie
// Alarm_0145	145	Error	Blokada dolnej pozycji siłownika chwytaka - sprawdź położenie ramienia lub usuń opakowanie
// Alarm_0146	146	Error	Brak opakowań w podajniku - dołóż opakownia lub sprawdź ich ułożenie

IF bAlarmInit THEN
    bAlarmInit := FALSE; 
	fbSourceInfo.Clear();
	fbSourceInfo.sName:=wsLiteral_TO_UTF8(sStationName);//'Machine';
	fbSourceInfo.nId:=udiStationID;//2700;
	// Alarm_0140	140	Error	Blokada otwarcia siłownika wjazdu opakowania - lewy - popraw lub usuń opakowanie
    arfbAlarm[0].CreateEx(stEventEntry := TC_EVENTS.AlarmClass.Alarm_0140, bWithConfirmation:= FALSE,  ipSourceInfo:= fbSourceInfo); 
	// Alarm_0141	141	Error	Blokada otwarcia siłownika wjazdu opakowania - prawy - popraw lub usuń opakowanie
	arfbAlarm[1].CreateEx(stEventEntry := TC_EVENTS.AlarmClass.Alarm_0141, bWithConfirmation:= FALSE,  ipSourceInfo:= fbSourceInfo); 
	// Alarm_0142	142	Error	Blokada lewej pozycji siłownika chwytaka - sprawdź położenie ramienia
	arfbAlarm[2].CreateEx(stEventEntry := TC_EVENTS.AlarmClass.Alarm_0142, bWithConfirmation:= FALSE,  ipSourceInfo:= fbSourceInfo); 
	// Alarm_0143	143	Error	Blokada prawej pozycji siłownika chwytaka - sprawdź położenie ramienia
	arfbAlarm[3].CreateEx(stEventEntry := TC_EVENTS.AlarmClass.Alarm_0143, bWithConfirmation:= FALSE,  ipSourceInfo:= fbSourceInfo); 
	// Alarm_0144	144	Error	Blokada górnej pozycji siłownika chwytaka - sprawdź położenie ramienia lub usuń opakowanie
	arfbAlarm[4].CreateEx(stEventEntry := TC_EVENTS.AlarmClass.Alarm_0144, bWithConfirmation:= FALSE,  ipSourceInfo:= fbSourceInfo); 
	// Alarm_0145	145	Error	Blokada dolnej pozycji siłownika chwytaka - sprawdź położenie ramienia lub usuń opakowanie
	arfbAlarm[5].CreateEx(stEventEntry := TC_EVENTS.AlarmClass.Alarm_0145, bWithConfirmation:= FALSE,  ipSourceInfo:= fbSourceInfo); 
	// Alarm_0146	146	Error	Brak opakowań w podajniku - dołóż opakownia lub sprawdź ich ułożenie
	arfbAlarm[6].CreateEx(stEventEntry := TC_EVENTS.AlarmClass.Alarm_0146, bWithConfirmation:= FALSE,  ipSourceInfo:= fbSourceInfo); 
END_IF


tonGate1Error			(IN:= NOT bSensorGate1				AND bGate1 									AND NOT bError, PT:=T#2S);
tonGate2Error			(IN:= NOT bSensorGate2				AND bGate2 									AND NOT bError, PT:=T#2S);	
tonArmLeftPositionError	(IN:= NOT bSensorArmLeft			AND bArmLeft 								AND NOT bError, PT:=T#2S);	
tonArmRightPostionError	(IN:= NOT bSensorArmRight			AND NOT bArmLeft 							AND NOT bError, PT:=T#2S);	
tonArmUpPositionError	(IN:= NOT bSensorArmUp				AND NOT bArmDown							AND NOT bError, PT:=T#2S);
tonArmDownPositionError	(IN:= (NOT bSensorArmDown			AND bArmDown		AND NOT bManualMode )	AND NOT bError, PT:=T#2S);
	
tonBottleAndFormTooLong	(IN:= NOT bSensorBottlePresent	AND NOT bError		AND bRun AND NOT bSimualtionMode, PT:=T#5M);//było 30s
tonEstopDelay			(IN:= bEStop,	PT:=T#3S);
bStateError				:= (eState = E_Station.eError OR eState = E_Station.eResetting);
	
IF (bEnable OR ((eState = E_Station.ePreparingToDisable) )) AND tonEstopDelay.Q THEN
	// Alarm_0140	140	Error	Blokada otwarcia siłownika wjazdu opakowania - lewy - popraw lub usuń opakowanie
	//Bląd siłownika wjazdu opakownia - lewy
	IF tonGate1Error.Q THEN
		IF NOT arfbAlarm[0].bActive THEN
			arfbAlarm[0].Raise(nTimeStamp:=0);
		END_IF
	ELSE	
		IF  arfbAlarm[0].bActive AND bReset THEN
			arfbAlarm[0].Clear(nTimeStamp:=0, bResetConfirmation:= FALSE);
		END_IF	
//		bError 								:= TRUE;
// 		udiErrorID							:=	101;
// 		//udiErrorID 							:=	udiErrorID;
// 		//udiErrorID 							:=	udiErrorID+iStationIndex; //+1100		
// 		sErrorDescription					:=	'Blokada otwarcia siłownika wjazdu opakowania - lewy - popraw lub usuń opakowanie';	
// 		sErrorDescription2					:=	'';			
	END_IF;
	// Alarm_0141	141	Error	Blokada otwarcia siłownika wjazdu opakowania - prawy - popraw lub usuń opakowanie
	//Bląd siłownika wjazdu opakownia - prawy
	IF tonGate2Error.Q THEN
		IF NOT arfbAlarm[1].bActive THEN
			arfbAlarm[1].Raise(nTimeStamp:=0);
		END_IF
	ELSE	
		IF  arfbAlarm[1].bActive AND bReset THEN
			arfbAlarm[1].Clear(nTimeStamp:=0, bResetConfirmation:= FALSE);
		END_IF	
// 		bError 								:= TRUE;
// 		udiErrorID							:=	102;
// 		//udiErrorID 							:=	udiErrorID+iStationIndex;
// 		sErrorDescription					:=	'Blokada otwarcia siłownika wjazdu opakowania - prawy - popraw lub usuń opakowanie';	
// 		sErrorDescription2					:=	'';			
	END_IF;
	// Alarm_0142	142	Error	Blokada lewej pozycji siłownika chwytaka - sprawdź położenie ramienia
	//Bląd siłownika ramienia - pozycja lewa
	IF tonArmLeftPositionError.Q THEN
		IF NOT arfbAlarm[2].bActive THEN
			arfbAlarm[2].Raise(nTimeStamp:=0);
		END_IF
	ELSE	
		IF  arfbAlarm[2].bActive AND bReset THEN
			arfbAlarm[2].Clear(nTimeStamp:=0, bResetConfirmation:= FALSE);
		END_IF	
// 		bError 								:= TRUE;
// 		udiErrorID							:=	103;
// 		//udiErrorID 							:=	udiErrorID+iStationIndex;
// 		sErrorDescription					:=	'Blokada lewej pozycji siłownika chwytaka - sprawdź położenie ramienia';	
// 		sErrorDescription2					:=	'';			
	END_IF;	
	// Alarm_0143	143	Error	Blokada prawej pozycji siłownika chwytaka - sprawdź położenie ramienia
	//Bląd siłownika ramienia - pozycja prawa
	IF tonArmRightPostionError.Q THEN
		IF NOT arfbAlarm[3].bActive THEN
			arfbAlarm[3].Raise(nTimeStamp:=0);
		END_IF
	ELSE	
		IF  arfbAlarm[3].bActive AND bReset THEN
			arfbAlarm[3].Clear(nTimeStamp:=0, bResetConfirmation:= FALSE);
		END_IF	
// 		bError 								:= TRUE;
// 		udiErrorID							:=	104;
// 		//udiErrorID 							:=	udiErrorID+iStationIndex;
// 		sErrorDescription					:=	'Blokada prawej pozycji siłownika chwytaka - sprawdź położenie ramienia';	
// 		sErrorDescription2					:=	'';			
	END_IF;	
	// Alarm_0144	144	Error	Blokada górnej pozycji siłownika chwytaka - sprawdź położenie ramienia lub usuń opakowanie
	//Bląd siłownika ramienia - pozycja górna
	IF tonArmUpPositionError.Q THEN
		IF NOT arfbAlarm[4].bActive THEN
			arfbAlarm[4].Raise(nTimeStamp:=0);
		END_IF
	ELSE	
		IF  arfbAlarm[4].bActive AND bReset THEN
			arfbAlarm[4].Clear(nTimeStamp:=0, bResetConfirmation:= FALSE);
		END_IF	
// 		bError 								:= TRUE;
// 		udiErrorID							:=	105;
// 		//udiErrorID 							:=	udiErrorID+iStationIndex;
// 		sErrorDescription					:=	'Blokada górnej pozycji siłownika chwytaka - sprawdź położenie ramienia lub usuń opakowanie';	
// 		sErrorDescription2					:=	'';			
	END_IF;	
	// Alarm_0145	145	Error	Blokada dolnej pozycji siłownika chwytaka - sprawdź położenie ramienia lub usuń opakowanie
	//Bląd siłownika ramienia - pozycja górna
	IF tonArmDownPositionError.Q THEN
		IF NOT arfbAlarm[5].bActive THEN
			arfbAlarm[5].Raise(nTimeStamp:=0);
		END_IF
	ELSE	
		IF  arfbAlarm[5].bActive AND bReset THEN
			arfbAlarm[5].Clear(nTimeStamp:=0, bResetConfirmation:= FALSE);
		END_IF		
	
// 		bError 								:= TRUE;
// 		udiErrorID							:=	106;
// 		//udiErrorID 							:=	udiErrorID+iStationIndex;
// 		sErrorDescription					:=	'Blokada dolnej pozycji siłownika chwytaka - sprawdź położenie ramienia lub usuń opakowanie';	
// 		sErrorDescription2					:=	'';			
	END_IF;			
	// Alarm_0146	146	Error	Brak opakowań w podajniku - dołóż opakownia lub sprawdź ich ułożenie		
	//Bląd braku opakowań w podajniku butelek
	IF tonBottleAndFormTooLong.Q THEN
		IF NOT arfbAlarm[6].bActive THEN
			arfbAlarm[6].Raise(nTimeStamp:=0);
		END_IF
	ELSE	
		IF  arfbAlarm[6].bActive AND bReset THEN
			arfbAlarm[6].Clear(nTimeStamp:=0, bResetConfirmation:= FALSE);
 		END_IF	
// 		bError 								:= TRUE;
// 		udiErrorID							:=	107;
// 		//udiErrorID 							:=	udiErrorID+iStationIndex;
// 		sErrorDescription					:=	'Brak opakowań w podajniku - dołóż opakownia lub sprawdź ich ułożenie';	
// 		sErrorDescription2					:=	'';			
	END_IF;	
	
//Rezerwa numerów udiErrorID: 108, 109, 110
ELSE
	bError := FALSE;
END_IF

//-----------------------------------------------------------------------
IF bError AND NOT bStateError THEN

	IF eLastState = eRunning THEN
		bCycleNotDone						:= TRUE;
	END_IF

	eState 									:= E_Station.eError;
END_IF

//------------------------------------------------------------------------

(*Wyświetlanie błedu na wyjściu*)
bError							:= FALSE;
FOR nAlarmNumerator := 0 TO 19 DO
	bError						:= bError OR arfbAlarm[nAlarmNumerator].bActive;
END_FOR

(*Przepisywanie nazwy stacji*)
sErrorStationName 							:= WSTRING_TO_STRING(sStationName);
END_ACTION

ACTION aHoming:
CASE iHomingStep OF
	0:
		iHomingStep				:=	iHomingStep	+	10;
                        		
	10:                 		
		bGripper 				:=	FALSE;
		iHomingStep				:=	iHomingStep	+	10;
                        	
	20:                 	
		bArmDown				:=	FALSE;
		IF bSensorArmUp THEN
				iHomingStep		:=	iHomingStep	+	10;
		END_IF
	30:

		bArmLeft				:=	FALSE;
		IF bSensorArmRight THEN
			iHomingStep			:=	iHomingStep +10;			
		END_IF

	40:
		bGate1					:=	FALSE;
		bGate2					:=	TRUE;		
		IF bSensorGate2 THEN
			iHomingStep			:=	iHomingStep +10;		
		END_IF

	50:
		bFormPositioning		:=	FALSE;
		IF bSensorFormPositioningClosed THEN
			iHomingStep			:=	iHomingStep +10;		
		END_IF
		
	60:
		eState					:=	E_Station.eHomingDone;
		eRunningState			:=	E_BottleFeederState.eReady;		
		iHomingStep				:=	0;
END_CASE
END_ACTION

ACTION aLimits:
IF tAllowFormDelay<T#700MS THEN
	tAllowFormDelay:=T#700MS;
END_IF

IF tSensorFormDelay<T#50MS THEN
	tSensorFormDelay:=T#300MS;
END_IF

IF tSensorBottleDelay<T#0MS THEN
	tSensorBottleDelay:=T#0MS;
END_IF

{warning 'dodać blokady w trybie manualnym żeby nie było kolicji'}
END_ACTION

ACTION aManualMovements:
IF NOT bRunPrepare AND NOT bRun THEN
	bGate1					:=		bManualGate1;			
	bGate2					:=		bManualGate2;			
	bArmDown				:=		bManualArmDown;			
	bArmLeft				:=		bManualArmLeft;			
	bGripper				:=		bManualGripper;			
	bFormPositioning		:=		bManualFormPositioning;		
ELSE
	bManualGate1			:=		FALSE;			
	//bManualGate2			:=		FALSE;		
	bManualArmDown			:=		FALSE;		
	bManualArmLeft			:=		FALSE;		
	bManualGripper			:=		FALSE;		
	bManualFormPositioning	:=		FALSE;	
END_IF

IF bHoming THEN 
	eState								:= E_Station.eHoming;
END_IF

IF NOT bEnable	THEN
	eState								:= E_Station.eReady;
END_IF

aRunning();

IF NOT bRun THEN

	bCycleDone					:= FALSE;
	bCycleNotDone				:= FALSE;
END_IF
END_ACTION

ACTION aResetCommands:

bGate1						:= FALSE;
bGate2						:= TRUE;
bGripper 					:= FALSE;
bArmDown					:= FALSE;
bArmLeft					:= FALSE;
bFormPositioning			:= FALSE;
                               
bManualGate1				:= FALSE;
bManualGate2				:= FALSE;	
bManualArmLeft				:= FALSE;
bManualArmDown				:= FALSE;
bManualGripper				:= FALSE;	
bManualFormPositioning		:= FALSE;
                               
iHomingStep					:= 0;
END_ACTION

ACTION aRunning:

CASE eRunningState OF

//--------------------------------------------------------------------------------------	
	//Pozycja gotowości 
	E_BottleFeederState.eReady:
	
		IF NOT bCycleDone AND NOT bCycleNotDone THEN	
			IF bRunPrepare OR bRun THEN
				eRunningState		:=	E_BottleFeederState.ePreparingToMove;
			END_IF
		END_IF
		
//--------------------------------------------------------------------------------------	
	//Przygotowanie do ruchu
	E_BottleFeederState.ePreparingToMove:
	
		bGripper 					:= FALSE;
		bGate1						:= FALSE;
		bGate2						:= TRUE;
		bArmDown					:= FALSE;
		bArmLeft					:= FALSE;
		bFormPositioning			:= FALSE;

		IF tonBottleSensorDelay.Q AND fbLevelSensor.bOut AND bRun AND bEstopAndDoors THEN
			eRunningState			:= E_BottleFeederState.eMoveToCatch;
		END_IF

		IF tonAllowEmptyForm.Q THEN
			IF tonFormsPresentDelay.Q  THEN
				eRunningState		:= E_BottleFeederState.eBackToPosition;			
			END_IF
		END_IF
		
//--------------------------------------------------------------------------------------		
	E_BottleFeederState.eCloseFirstGate:
		;
		
//--------------------------------------------------------------------------------------	
	E_BottleFeederState.eMoveToCatch:
	
		bGripper 					:=	 FALSE;
		bGate1						:=	 FALSE;
		bGate2						:=	 TRUE;
		bArmDown					:=	 FALSE;
		bArmLeft					:=	 TRUE;
		bFormPositioning			:=	 FALSE;
	
		IF bSensorArmLeft THEN 
			eRunningState			:=	E_BottleFeederState.eCloseGripper;
		END_IF
		
//-------------------------------------------------------------------------------------		

	E_BottleFeederState.eCloseGripper:
	
		bGripper					:=	TRUE;
		IF tonGripper.Q THEN
			eRunningState			:=	E_BottleFeederState.eGoAbove;
		END_IF
	
	E_BottleFeederState.eOpenSecondGate:
		
		;
		
	E_BottleFeederState.eGoAbove:

		bGripper 					:=	 TRUE;
		bGate1						:=	 TRUE;
		bGate2						:=	 FALSE;
		bArmDown					:=	 FALSE;
		bArmLeft					:=	 FALSE;
		bFormPositioning			:=	 FALSE;
		
		IF bSensorArmRight AND tonFormsPresentDelay.Q THEN
			eRunningState			:=	E_BottleFeederState.eCloseSecondGate;			
		END_IF
	
//--------------------------------------------------------------------------------------
	E_BottleFeederState.eCloseSecondGate:	
	
		bGripper 					:=	 TRUE;
		bGate1						:=	 FALSE;
		bGate2						:=	 TRUE;
		bArmDown					:=	 FALSE;
		bArmLeft					:=	 FALSE;
		bFormPositioning			:=	 FALSE;
		eRunningState				:=	E_BottleFeederState.eCloseStoper;	
		
//----------------------------------------

	E_BottleFeederState.eCloseStoper:		
	
		bFormPositioning			:=	TRUE;
		//IF  (NOT bSensorFormAfterPresent OR bManualMode) THEN
			eRunningState			:=	E_BottleFeederState.eInsterting;			
		//END_IF	

//------------------------------------------------------------------------------------	
	// Włóż butelek
	E_BottleFeederState.eInsterting:
	
		bArmDown						:=	TRUE;
		IF	(ftIbSensorLifterDown.Q OR bSensorArmDown) OR NOT bArmDown THEN //Przeleciało przez czujnik albo jest	
			eRunningState					:=	E_BottleFeederState.eOpenGripper;	
		END_IF
//------------------------------------------------------------------------------------		
	// Otwórz chwytak 
	E_BottleFeederState.eOpenGripper:
	
		IF tonArmDown.Q THEN 
			bGripper					:=	FALSE;
		END_IF
		
		IF tonOpenedGripper.Q  THEN 
			eRunningState			:=	E_BottleFeederState.eBackToPosition;	
		END_IF

//-----------------------------------------------------------------------------------	
	// Powrót do pozycji gotowości
	E_BottleFeederState.eBackToPosition:
	
		bArmDown						:=	FALSE;
		bFormPositioning				:=	FALSE;
		
		IF bSensorArmUp THEN
			bCycleDone				:=	TRUE;	
			eRunningState			:=	E_BottleFeederState.eReady;	
		END_IF

END_CASE
END_ACTION

ACTION aSignals:

	tonPreparingToDisabled	(IN:= eState = E_Station.ePreparingToDisable, 			PT:= T#1S);
	tonPreparingToReadyOn	(IN:= eState = E_Station.ePreparingToReady, 			PT:= T#300MS);
	tofRunning				(IN:= eState = E_Station.eRunning, 						PT:= T#10S);	

	tonBottleSensorDelay	(IN:= bSensorBottlePresent OR (bRun AND bManualMode) OR bSimulationSensor,	PT:=tSensorBottleDelay);
	tonAllowEmptyForm 		(IN:= (NOT bSensorBottlePresent OR NOT  fbLevelSensor.bOut OR NOT bEstopAndDoors) AND bSensorFormPresent AND
								eRunningState = E_BottleFeederState.ePreparingToMove AND
								eState = E_Station.eRunning,
																			 		PT:=tAllowFormDelay);							
	
	tonFormsPresentDelay	(IN:= bSensorFormPresent OR (bRun AND bManualMode), 	PT:=tSensorFormDelay);

	ftIbSensorLifterDown	(CLK:= bSensorArmDown,									Q=>);

	rtResetCycle			(CLK:= bResetCycle);
	tonGripper				(IN:= bGripper,											PT:=T#80MS);
	tonOpenedGripper		(IN:= NOT bGripper,										PT:=T#10MS);
	tonArmDown				(IN:= bArmDown, 										PT:=T#230MS);
	





	bSimulationSensor	:=	bSimualtionMode AND NOT tonBottleSensorDelay.Q;
END_ACTION

ACTION aStationID:
udiStationID	:=	iStationIndex;
END_ACTION

ACTION aStatistic:

//Statystyka do zliczania czasu cyklu 
rtrigCycleTimerRead(CLK:=bCycleDone);

	IF rtrigCycleTimerRead.Q THEN
		tCycleTime:=tonCycleTimer.ET;
	END_IF
	
tonCycleTimer(IN:= eRunningState<>E_BottleFeederState.eReady AND eRunningState<>E_BottleFeederState.ePreparingToMove , PT:=T#1D);
END_ACTION

ACTION aStatus:

(*Zapisywanie ostatniego stanu*)
	IF eLastStateTemp<>eState THEN
		eLastState := eLastStateTemp;
	END_IF
	eLastStateTemp := eState;
	
	IF eLastRunningStateTemp<>eRunningState THEN
		eLastRunningState := eLastRunningStateTemp;
	END_IF
	eLastRunningStateTemp := eRunningState;
(*Koniec Zapisywanie ostatniego stanu*)
END_ACTION

ACTION aWarnings:

//Filtrowanie czujnika ultradźwiękowego

fbLevelSensor	(bIN:= bLevelSensor AND tofRunning.Q, tFilterTimeOn:= T#2S, tFilterTimeOff:=T#5S , bOUT=> );

IF NOT fbLevelSensor.bOUT THEN
	bWarning1						:=	TRUE;			
	udiWarningID					:=	1;
	sWarning1Description			:=	'Niski poziom butelek w sorterze butelek';
ELSE
	bWarning1						:=	FALSE;			
	udiWarningID					:=	0;
	sWarning1Description			:=	'';
END_IF

IF tofRunning.Q AND NOT bEstopAndDoors THEN
	bWarning2						:=	TRUE;	
	sWarning2Description			:=	'Otwarte drzwi';
ELSE
	bWarning2						:=	TRUE;	
	sWarning2Description			:=	'';
END_IF
END_ACTION

END_FUNCTION_BLOCK

// ---- POUs/FB/FB_SpringGateV2.TcPOU
(*
Nazwa:			FB_SpringGate
Opis:			Stacja szlabanów do zatrzymywania formatek 
Wersja:			v1.0
Data:			2018-10-31
Autor:			DP
Urzadzenia:		do 2 szlabanów i czujniki zamkniecia/otwarcia
Konfiguracja:	
Info: 
- zmiana 3 / nie wylaczenia szlabanow w disabled
- opcja wpusc/wypuść
- czasy na wjazd i wyjazd formatek
*)
FUNCTION_BLOCK FB_SpringGateV2
VAR_INPUT
	bEnable: BOOL;						//Zezwolenie na pracę
	bEStop:BOOL;						//Stop Awaryjny włączony
	bRun:BOOL;							//Rozkaz wpuszczenia dwóch formatek 
	bHoming:BOOL;						//Zezwolenie na wykonanie bazowania i pozycjonowania podajnika
	bHeightSet:BOOL;					//Ustaw wysokość
	bIgnoreError:BOOL;					//Ignorowania błędów cyklu pracy
	bReset:BOOL;						//Reset błędu, jeśli w stanie "eError"
	bOpenedGate1ActuatorSensor:BOOL;	//Czujnik otwarcia siłownika szlabanu 1
	bClosedGate1ActuatorSensor:BOOL;	//Czujnik zamknięcia siłownika szlabanu 1
	bFullBadBottleConveyorSensor:BOOL;	//Zapełniony transporter odrzuconych butelek
	bManualMovement:BOOL;				//Zezwolenie na ruchy ręcznę
	nTimeInserting:UINT;			//Czas na wpuszczenie formatek
	bHomingStateGate1:BOOL;				//Stan bazowania szlabanów nr 1
	bResetState:BOOL;					//Resetowanie stanu stacji
	_ALARMINFO_ :BOOL;
	iStationIndex:UDINT;				//Numer stacji 
	sStationName:WSTRING;				//Nazwa stacji

END_VAR
VAR_OUTPUT
	
	eState: E_Station;						//Stan ogólny bloku
	eRunningState: E_EntranceGatesState;	//Stan szlabanów
	bError: BOOL;							//Błąd stacji	
	nErrorNr: UDINT;						//Nr błędu podajnika platynek
	sErrorDescription:STRING(200);				//Opis błędu
	sErrorDescription2:STRING(200);				//Opis błędu
	sErrorStationName:STRING;				//Nazwa stacji
	udiStationID:UDINT;						//Nr stacji	
	bGate1Actuator:BOOL;					//Sterownie siłownika szlabanu 1
	tCycleTime:TIME;
	bHomingDone:BOOL;						//Wymagane ponowne bazowanie (blad podczas bazowania lub stop awaryjny)
	bCycleDone:BOOL;
	bCycleNotDone:BOOL;
END_VAR

VAR

// Timer blokady otwierania chwytaka
	tonOpeningGate1Blocked: TON;
	tonClosingGate1Blocked: TON;	
	tonCycleTimer:TON;
	rtrigCycleTimerRead:R_TRIG;	
	bLastStateGate1Actuator: BOOL;
	
	eLastState: E_Station;							//Stan ogólny bloku
	eLastRunningState: E_EntranceGatesState;		//Stan podbloku
	eLastStateTemp: E_Station;						//Stan ogólny bloku
	eLastRunningStateTemp: E_EntranceGatesState;	//Stan podbloku
	tonFullBadBottleConveyor: TON;
	bStateError: BOOL;
	tonInserting: TON;
	
	//Zmienne od EVENTLOGGER
	bAlarmInit 						: BOOL := TRUE; 
	nAlarmNumerator					: INT;
	arfbAlarm						: ARRAY[0..19] OF  FB_TcAlarm;		//Tablica bloczków błędów
	fbSourceInfo 					: FB_TcSourceInfo;
	iSourceInfo						: I_TcSourceInfo;
	sAlarmTest						: STRING;
	//Koniec zmiennych od EVENTLOGGER
	
END_VAR

VAR_IN_OUT
	bManualGate1Actuator:BOOL;			//Ruch ręczny siłownikiem szlabanu 1
END_VAR

(*Przepisywanie Homingu , rozdzielenie wyjść*)

ErrorHandling();
Control();
Statistics();
aStationID();

(*Zapisywanie ostatniego stanu*)
IF eLastStateTemp<>eState THEN
	eLastState := eLastStateTemp;
END_IF
eLastStateTemp := eState;
IF eLastRunningStateTemp<>eRunningState THEN
	eLastRunningState := eLastRunningStateTemp;
END_IF
eLastRunningStateTemp := eRunningState;
(*Koniec Zapisywanie ostatniego stanu*)


IF bResetState THEN
	bGate1Actuator:=bHomingStateGate1;
END_IF

ACTION aStationID:
udiStationID	:=	iStationIndex;
END_ACTION

ACTION Control:

	(** TIMERY**)
	tonInserting(IN:=eRunningState=E_EntranceGatesState.ePulling, PT:=UINT_TO_TIME(nTimeInserting));

	
	(*****Wyłączenie enable*****)
	IF NOT bEnable THEN
		IF eState <> E_Station.eDisabled AND eState <> E_Station.ePreparingToDisable THEN
				eState 				:= E_Station.ePreparingToDisable; 
		END_IF	
	END_IF

	(*****Estop*****)
	IF NOT bEstop  THEN	
		IF eState <> E_Station.eAborted AND eState <> E_Station.eAborting AND eState <> E_Station.eDisabled THEN
				eState 				:= E_Station.eAborting; 
		END_IF
	END_IF

	
	CASE eState OF
	/////////////////////////////	
		E_Station.eDisabled: 					// Stan nieaktywnosci (Stacja wyłączona) 
			bGate1Actuator			:=FALSE;
			IF bEnable THEN
				eState 				:= E_Station.ePreparingToReady; 
			END_IF 
			
    /////////////////////////////	    
		E_Station.eAborted: 					// Stan bezpiecznego zatrzymania (po Abortingu) 

			IF bEStop THEN
				eState 				:= E_Station.ePreparingToReady;
			END_IF
			
	/////////////////////////////	
		E_Station.eAborting:                 	// Stan bezpiecznego zatrzymywania (po EStopie)
		
			//bGate1Actuator			:=	FALSE;
			eState 					:=	E_Station.eAborted;  
			eRunningState			:=	E_EntranceGatesState.eDisabled;
			
	/////////////////////////////			
		E_Station.eError:                 	 	// Stan błędu 	
	
			IF bReset THEN
				eState 				:= E_Station.eResetting;
				
			END_IF
			
	/////////////////////////////
		E_Station.eResetting:					// Stan resetowania bledu (po Errorze)
			
			bError := FALSE;
			IF NOT bError THEN
				nErrorNr 			:=	0;
   				sErrorDescription 	:=	'';
				eState 				:=	E_Station.ePreparingToReady;
			ELSE
				eState 				:=	E_Station.eError;
			END_IF
        
	/////////////////////////////
		E_Station.eManualMovement:     			// Stan ruchów manualnych  
       
			ManualMovements();
			//Wyjście z trybu serwisowego
			IF NOT bManualMovement THEN
				bGate1Actuator				:=	bLastStateGate1Actuator;
				eState:=E_Station.eReady;
			END_IF

	/////////////////////////////
		E_Station.eHoming:						// Stan bazowania 

			Homing();
			IF NOT bHoming AND NOT bHeightSet THEN
			   eState:=E_Station.ePreparingToReady;
			END_IF		
			
	/////////////////////////////
		E_Station.eHomingDone:                  // Stan wykonania bazowania 
		
			//bGate1Actuator					:=	FALSE;
			bHomingDone							:=	TRUE;
			IF NOT bHoming AND NOT bHeightSet THEN
			   eState:=E_Station.eReady;
			END_IF
			
	/////////////////////////////
		E_Station.ePreparingToReady:            // Stan przygotowywania do gotowosci (zawsze przed Ready)  
		
         	bGate1Actuator						:=TRUE;
			eRunningState						:=E_EntranceGatesState.eReady;
			eState								:=E_Station.eReady;	
			
	/////////////////////////////
		E_Station.ePreparingToDisable:          // Stan przygotowywania do nieaktywnosci (po wyłączeniu Enable) 
  
			bGate1Actuator						:=FALSE;		
			eState								:=E_Station.eDisabled;
			eRunningState						:=E_EntranceGatesState.eDisabled;
			
	/////////////////////////////
		E_Station.eReady:						// Stan gotowosci 

			IF bRun AND NOT bCycleDone AND NOT bCycleNotDone THEN
				eState 				:= E_Station.eStarting; 
			END_IF
			IF bHoming OR bHeightSet THEN
				eState 				:= E_Station.eHoming; 
			END_IF
			IF bManualMovement THEN
				//Jeśli przejście w tryb ruchów manualnych przepisz wszystkie stany siłowników sterowanych przez moduł
				//aby zapobiec ewentualnym kolizjom po wejściu w tryb serwisowy
				bLastStateGate1Actuator		:=	bGate1Actuator;
				bManualGate1Actuator		:=	bGate1Actuator;
				eState 						:=	E_Station.eManualMovement; 
			END_IF
			IF NOT bRun THEN
				bCycleDone 					:= FALSE;
				bCycleNotDone 				:= FALSE;			
			END_IF
			
	/////////////////////////////
		E_Station.eStopping:					// Stan zatrzymywania 
			
			Running();
			
			bGate1Actuator 					:=	TRUE;
			eRunningState					:=	E_EntranceGatesState.eReady;
			eState 							:=	E_Station.eReady;	
			
	/////////////////////////////
		E_Station.eStarting:                  	// Stan uruchamiania (po Ready)
		
			eState					 := E_Station.eRunning; 
			eRunningState			:=E_EntranceGatesState.eReady;
				
	/////////////////////////////
		E_Station.eRunning:               		// Stan wykonywania cyklu (po Startingu), w tym stanie osobny
 
			Running();
			IF NOT bRun THEN					(*Przerywanie cyklu*)
				eState 				 := E_Station.eStopping;	
			END_IF
			//IF bCycleDone OR bCycleNotDone THEN (*Cykl zakończony*)
			//	eState 				 := E_Station.eReady;	
			//END_IF	
			
	/////////////////////////////		
	END_CASE
END_ACTION

ACTION ErrorHandling:
// Alarm_0160	160	Error	Blokada otwarcia szlabanu wjazdowego nr 1 - sprawdź czujnik lub odblokuj mechanicznie
// Alarm_0161	161	Error	Blokada zamknięcia szlabanu wjazdowego nr 1 - sprawdź czujnik lub odblokuj mechanicznie

IF bAlarmInit THEN
    bAlarmInit := FALSE; 
	fbSourceInfo.Clear();
	fbSourceInfo.sName:=wsLiteral_TO_UTF8(sStationName);//'Machine';
	fbSourceInfo.nId:=iStationIndex;//2700;
	// Alarm_0160	160	Error	Blokada otwarcia szlabanu wjazdowego nr 1 - sprawdź czujnik lub odblokuj mechanicznie
	arfbAlarm[0].CreateEx(stEventEntry := TC_EVENTS.AlarmClass.Alarm_0160, bWithConfirmation:= FALSE,  ipSourceInfo:= fbSourceInfo); 
	// Alarm_0161	161	Error	Blokada zamknięcia szlabanu wjazdowego nr 1 - sprawdź czujnik lub odblokuj mechanicznie
	arfbAlarm[1].CreateEx(stEventEntry := TC_EVENTS.AlarmClass.Alarm_0161, bWithConfirmation:= FALSE,  ipSourceInfo:= fbSourceInfo); 
END_IF



//OBSŁUGA BŁĘDÓW PODAJNIKA PLATYNEK

//************LISTA BŁĘDÓW***************
bStateError:= (eState=E_Station.eError) OR (eState=E_Station.eResetting);

IF bEnable THEN
	
	// Alarm_0160	160	Error	Blokada otwarcia szlabanu wjazdowego nr 1 - sprawdź czujnik lub odblokuj mechanicznie
	//Error 1 - Blokada otwarcia szlabanu wejściowego nr 1
	tonOpeningGate1Blocked(IN:= bGate1Actuator AND NOT bOpenedGate1ActuatorSensor, PT:=T#2S);
	IF tonOpeningGate1Blocked.Q THEN
		IF NOT arfbAlarm[0].bActive THEN
			arfbAlarm[0].Raise(nTimeStamp:=0);
		END_IF
	ELSE	
		IF  arfbAlarm[0].bActive AND bReset THEN
			arfbAlarm[0].Clear(nTimeStamp:=0, bResetConfirmation:= FALSE);
		END_IF	
// 		sErrorDescription:='Blokada otwarcia szlabanu wjazdowego nr 1 - sprawdź czujnik lub odblokuj mechanicznie';
// 		bError := TRUE;
// 		nErrorNr:=111;	
// 		//nErrorNr:=nErrorNr+iStationIndex;
	END_IF

	// Alarm_0161	161	Error	Blokada zamknięcia szlabanu wjazdowego nr 1 - sprawdź czujnik lub odblokuj mechanicznie	
	//Error 2 - Blokada zamknięcia szlabanu wejściowego nr 1
	tonClosingGate1Blocked(IN:= NOT bGate1Actuator AND NOT bClosedGate1ActuatorSensor, PT:=T#2S);
	IF tonClosingGate1Blocked.Q THEN
		IF NOT arfbAlarm[1].bActive THEN
			arfbAlarm[1].Raise(nTimeStamp:=0);
		END_IF
	ELSE	
		IF  arfbAlarm[1].bActive AND bReset THEN
			arfbAlarm[1].Clear(nTimeStamp:=0, bResetConfirmation:= FALSE);
		END_IF	
// 		sErrorDescription:='Blokada zamknięcia szlabanu wjazdowego nr 1 - sprawdź czujnik lub odblokuj mechanicznie';
// 		bError := TRUE;
// 		nErrorNr:=112;	
// 		//nErrorNr:=nErrorNr+iStationIndex;
	END_IF
	
//Rezerwa numerów udiErrorID: 113, 114, 115, 116, 117, 118, 119, 120,
ELSE
	bError := FALSE;
END_IF

//*******KONIEC LISTA BŁĘDÓW***************	



	

//******************PRZEJŚCIE DO eERROR*****************************

IF bError AND NOT bStateError THEN
	IF eLastState = eRunning THEN
		bCycleNotDone := TRUE;
	END_IF
	eState := E_Station.eError;
END_IF

//****************WYŚWIETLANIE STATUSU BLEDU***********************



(*Wyświetlanie błedu na wyjściu*)
bError							:= FALSE;
FOR nAlarmNumerator := 0 TO 19 DO
	bError						:= bError OR arfbAlarm[nAlarmNumerator].bActive;
END_FOR


(*Przepisywanie nazwy stacji*)
sErrorStationName:=WSTRING_TO_STRING(sStationName);
END_ACTION

ACTION Homing:
//BAZOWANIE SZLABANÓW
	
	bGate1Actuator:=bHomingStateGate1;
	// Jezeli bazowanie zostanie zakończone
	

	eState:=E_Station.eHomingDone;
END_ACTION

ACTION ManualMovements:

//W trybie ruchów manualnych wykonuj ruchy za pomocą rozkazów manualnych
//IF NOT bRun THEN
	bGate1Actuator:=bManualGate1Actuator;
//ELSE	//Kasuje zeby po cyklu nic sie nie poruszało
//	bGate1Actuator := FALSE;
//END_IF

	

IF bHoming OR bHeightSet THEN
	eState:=E_Station.eHoming;
END_IF
	
//Running();

IF NOT bRun THEN
	bCycleDone 					:= FALSE;
	bCycleNotDone 				:= FALSE;	
END_IF
END_ACTION

ACTION Running:


CASE eRunningState OF
	
	//NIEGOTOWY
	E_EntranceGatesState.eDisabled:
			eRunningState:=E_EntranceGatesState.eReady;
		
	//ZGRZEWANIE GOTOWY DO PRACY
	E_EntranceGatesState.eReady:
		
		//Jeśli komenda podania platynki przejdź do stanu zasysania platynki
		IF NOT bCycleDone AND NOT bCycleNotDone THEN
			IF bRun THEN
				eRunningState	:=E_EntranceGatesState.ePulling;
			END_IF
		END_IF

	//STAN BLOKOWANIA 

	//WSUWANIE NA TRANSPORTER
	E_EntranceGatesState.ePulling:
	
		bGate1Actuator 			:= FALSE;
		IF tonInserting.Q THEN
	 		eRunningState		:=	E_EntranceGatesState.ePullingDone;
		END_IF;
		 
	E_EntranceGatesState.ePullingDone:
		bCycleDone				:=	TRUE;
		IF NOT bRun THEN
			bGate1Actuator 			:= TRUE;
			eRunningState			:=	E_EntranceGatesState.eReady;

		END_IF
	

END_CASE
END_ACTION

ACTION Statistics:



rtrigCycleTimerRead(CLK:=eRunningState=E_EntranceGatesState.eReady);
IF rtrigCycleTimerRead.Q THEN
	tCycleTime:=tonCycleTimer.ET;
END_IF
tonCycleTimer(IN:=eRunningState>E_EntranceGatesState.eReady,PT:=T#1D);
END_ACTION

END_FUNCTION_BLOCK

// ---- POUs/P16_LabelMachine.TcPOU
(*
Nazwa:			P16_LabelMachine
Opis:			Stacja etykieciarki
Wersja:			v0.1
Data:			2018-10-10
Autor:			DP
Urzadzenia:		
Konfiguracja:	
Info:
Zmiany:
- 20231215 [DP] ServiceMode do czujnika przepełnienia etykieciarki

*)
PROGRAM P16_LabelMachine
VAR_INPUT
	IbLabelMachineFullSensor AT %I*: BOOL;	(*PLC.G1 robot*)	// Czujnik przepelnienia butelek na etykieciarce
END_VAR
VAR
	
	(************ETYKIECIARKA*******************)
	IbLabelMachineWorking AT %I*:BOOL;		(*PLC.A8*)			// Etykieciarka praca
	IbLabelMachineNotError AT %I*:BOOL;		(*PLC.A8*)			// Etykieciarka awaria
	QbLabelMachineStart AT %Q*:BOOL;		(*PLC.A20*)
	QbLabelMachineStop  AT %Q*:BOOL;
	// Czas wyłaczania etykieciarki
	tpLabelStop: TP;
	tpLabelStartDelay: TP;
	tonLabelStopError: TON;
	tonLabelMachineFullSensor: TON;
	tonLabelMachineFullSensorInfo: TON;	
	
	
	//Zmienne od EVENTLOGGER
	bAlarmInit 						: BOOL := TRUE; 
	nAlarmNumerator					: INT;
	arfbAlarm						: ARRAY[0..19] OF  FB_TcAlarm;		//Tablica bloczków błędów
	fbSourceInfo 					: FB_TcSourceInfo;
	iSourceInfo						: I_TcSourceInfo;
	sAlarmTest						: STRING;
	//Koniec zmiennych od EVENTLOGGER
END_VAR

aLabelMachine();

ACTION aLabelMachine:
// Alarm_0120	120	Error	Etykieciarka | Błąd - sprawdź urządzenie
// Alarm_0121	121	Error	Etykieciarka | Błąd załączenia - brak sygnału potwierdzenia pracy. Może być zablokowana przez system wizyjny - sprawdź urządzenie
// Alarm_0122	122	Error	Etykieciarka | Zapełniony transporter - sprawdź czujnik


IF bAlarmInit THEN
    bAlarmInit := FALSE; 
	fbSourceInfo.Clear();
	fbSourceInfo.sName:='Błąd systemu';
	fbSourceInfo.nId:=80;
	// Alarm_0120	120	Error	Etykieciarka | Błąd - sprawdź urządzenie
    arfbAlarm[0].CreateEx(stEventEntry := TC_EVENTS.AlarmClass.Alarm_0120, bWithConfirmation:= FALSE,  ipSourceInfo:= fbSourceInfo); 
	// Alarm_0121	121	Error	Etykieciarka | Błąd załączenia - brak sygnału potwierdzenia pracy. Może być zablokowana przez system wizyjny - sprawdź urządzenie
	arfbAlarm[1].CreateEx(stEventEntry := TC_EVENTS.AlarmClass.Alarm_0121, bWithConfirmation:= FALSE,  ipSourceInfo:= fbSourceInfo); 
	// Alarm_0122	122	Error	Etykieciarka | Zapełniony transporter - sprawdź czujnik
	arfbAlarm[2].CreateEx(stEventEntry := TC_EVENTS.AlarmClass.Alarm_0122, bWithConfirmation:= FALSE,  ipSourceInfo:= fbSourceInfo); 
END_IF



//Wywoływanie błędu etykieciarki

//BŁĄD 77  - Błąd ogólny etykieciarki
(*IF (P00_PackML.fbPMLAuto.ePMLState = E_PMLState.ePMLState_STARTING OR P00_PackML.fbPMLAuto.ePMLState = E_PMLState.ePMLState_EXECUTE) AND NOT IbLabelMachineNotError AND NOT VIS.bErrorOccure AND bLabelMachineCmdStart THEN
	bLabelMachineCmdStart														:= FALSE;
	LabelMachineError.bError													:= TRUE;
	LabelMachineError.nErrorCode												:= 77;
	LabelMachineError.bReset													:= FALSE;
	LabelMachineError.sErrorString												:= 'Etykieciarka | Błąd - sprawdź urządzenie';
	LabelMachineError.sErrorString2												:= '';
	LabelMachineError.sStationName												:= 'Błąd systemu';
*)
// Alarm_0121	121	Error	Etykieciarka | Błąd załączenia - brak sygnału potwierdzenia pracy. Może być zablokowana przez system wizyjny - sprawdź urządzenie
//BŁĄD 78  - brak sygnału pracy	
IF tonLabelStopError.Q AND NOT VIS.bErrorOccure AND bLabelMachineCmdStart THEN
	IF NOT arfbAlarm[1].bActive THEN
			bLabelMachineCmdStart														:= FALSE;
			arfbAlarm[1].Raise(nTimeStamp:=0);
		END_IF
	ELSE	
		IF  arfbAlarm[1].bActive AND LabelMachineError.bReset THEN
			arfbAlarm[1].Clear(nTimeStamp:=0, bResetConfirmation:= FALSE);
		END_IF	
//	bLabelMachineCmdStart														:= FALSE;
// 	LabelMachineError.bError													:= TRUE;
// 	LabelMachineError.nErrorCode												:= 78;
// 	LabelMachineError.bReset													:= FALSE;
// 	LabelMachineError.sErrorString												:= 'Etykieciarka | Błąd załączenia - brak sygnału potwierdzenia pracy. Może być zablokowana przez system wizyjny - sprawdź urządzenie';
// 	LabelMachineError.sErrorString2												:= '';
// 	LabelMachineError.sStationName												:= 'Błąd systemu';
END_IF
// Alarm_0122	122	Error	Etykieciarka | Zapełniony transporter - sprawdź czujnik
//BŁĄD 79  - zapełnienie etykieciarki 
IF tonLabelMachineFullSensor.Q AND NOT VIS.bErrorOccure THEN 
		IF NOT arfbAlarm[2].bActive THEN
			bLabelMachineCmdStart														:= FALSE;
			arfbAlarm[2].Raise(nTimeStamp:=0);
		END_IF
	ELSE	
		IF  arfbAlarm[2].bActive AND LabelMachineError.bReset THEN
			arfbAlarm[2].Clear(nTimeStamp:=0, bResetConfirmation:= FALSE);
		END_IF	
// 	bLabelMachineCmdStart														:= FALSE;
// 	LabelMachineError.bError													:= TRUE;
// 	LabelMachineError.nErrorCode												:= 79;
// 	LabelMachineError.bReset													:= FALSE;
// 	LabelMachineError.sErrorString												:= 'Etykieciarka | Zapełniony transporter - sprawdź czujnik';
// 	LabelMachineError.sErrorString2												:= '';
// 	LabelMachineError.sStationName												:= 'Błąd systemu';		
END_IF

// IF LabelMachineError.bError AND LabelMachineError.bReset THEN 
// 	
// 	LabelMachineError.bError													:= FALSE;
// 	LabelMachineError.nErrorCode												:= 0;
// 	LabelMachineError.bReset													:= FALSE;
// 	LabelMachineError.sErrorString												:= '';
// 	LabelMachineError.sErrorString2												:= '';
// 	LabelMachineError.sStationName												:= '';
// END_IF	
//ELSIF VIS.bErrorOccure THEN
IF LabelMachineError.bError	 THEN
	bLabelMachineCmdStart 														:= FALSE;
END_IF

(*Wyświetlanie błedu na wyjściu*)
LabelMachineError.bError							:= FALSE;
FOR nAlarmNumerator := 0 TO 19 DO
	LabelMachineError.bError						:= LabelMachineError.bError OR arfbAlarm[nAlarmNumerator].bActive;
END_FOR

//Timer błedu załączenia
//tonLabelStopError(IN:=	(P00_PackML.fbPMLAuto.ePMLState = E_PMLState.ePMLState_STARTING OR P00_PackML.fbPMLAuto.ePMLState = E_PMLState.ePMLState_EXECUTE) AND
//						bLabelMachineCmdStart AND NOT IbLabelMachineWorking AND NOT QbLabelMachineStart,PT:=T#500MS);
						
tonLabelStopError(IN:=	(P00_PackML.fbPMLAuto.ePMLState = E_PMLState.ePMLState_STARTING OR P00_PackML.fbPMLAuto.ePMLState = E_PMLState.ePMLState_EXECUTE) AND
						bLabelMachineCmdStart AND NOT IbLabelMachineWorking,PT:=T#10M);	//bylo 20s					
						
tpLabelStartDelay(IN:=IbEmergencyStop AND NOT LabelMachineError.bError AND bLabelMachineCmdStart ,PT:=T#500MS);//2s

//Sterowanie etykieciarką										// Nie w serwisie, bo w trybie serwisowym, był bład
tonLabelMachineFullSensor	(IN:=IbEmergencyStop AND IbLabelMachineFullSensor (*AND bLabelMachineEnable*) AND NOT VIS.bServiceMode AND 
								(P00_PackML.fbPMLAuto.ePMLState = E_PMLState.ePMLState_STARTING OR P00_PackML.fbPMLAuto.ePMLState = E_PMLState.ePMLState_EXECUTE OR P00_PackML.fbPMLAuto.ePMLState = E_PMLState.ePMLState_STOPPING)
								,PT:=T#8M); // zmiana z 7s i wykomentowe cmdStart
//Wykorzystywane 
tonLabelMachineFullSensorInfo	(IN:=IbLabelMachineFullSensor,PT:=T#2S); // WYkorzystywane do informacji

//QbLabelMachineStart 				:= tpLabelStartDelay.Q OR VIS.bLabelMachine1ManualStart;
QbLabelMachineStart 				:= IbEmergencyStop AND NOT LabelMachineError.bError AND bLabelMachineCmdStart;

(*Manual*)
IF NOT  (P00_PackML.fbPMLModeManager.eModeStatus = E_PMLUnitMode.ePMLUnitMode_MANUAL) THEN
	VIS.bLabelMachine1ManualStart												:= FALSE;
END_IF

(*Po stopie awaryjnym wyłączanie etykieciarki*)
IF NOT IbEmergencyStop THEN
	bLabelMachineCmdStart														:= FALSE;
	VIS.bLabelMachine1ManualStart												:= FALSE;
END_IF
END_ACTION

END_PROGRAM

// ---- POUs/P06_LidFeeder.TcPOU
PROGRAM P06_LidFeeder
VAR_INPUT
	IbLidFeederDragHomingSensor 			AT %I*  : BOOL;				// Czujnik bazowania
	IbLidFeederDragUpSensor 			 	AT %I*  : BOOL;				// Czujnik
	IbLidFeederDragDownSensor 				AT %I*  : BOOL;				// Czujnik
	IbLidFeederDragLeadBefore1UpSensor 		AT %I*  : BOOL;				// Czujnik
	IbLidFeederUpSensor1 					AT %I*	: BOOL; 								// Czujnik pozycji górnej ssawki podajnika platynek
	IbLidFeederUpSensor2 					AT %I*	: BOOL;
	IbLidFeederDownSensor1 					AT %I*	: BOOL;								
	IbLidFeederDownSensor2 					AT %I*	: BOOL;								
	IbLidFeederLowLevelSensor1  			AT %I* 	: BOOL;	
	IbLidFeederLowLevelSensor2  			AT %I* 	: BOOL;
	IbLidFeederFormPositioning1HideSensor			AT %I*	: BOOL; 
	IbLidFeederFormPositioning2HideSensor			AT %I*	: BOOL;
	IbLidFeederFirstFormSensorBeforeDrag			AT %I*	:BOOL;
	IbLidFeederSuckerSensor 				AT %I*	: BOOL;
	IbLidFeeder2SuckerSensor 				AT %I*	: BOOL;  
	bMovetoEndPositionLidFeeder				:BOOL;	
	QbLidFeederDragActuator                	  		: BOOL;				// Siłownikiem przeciągania (1 faza)					

END_VAR
VAR
	//Podajnik platynek
	fbLidFeeder										: FB_LidFeeder; 						// Blok sterowania podajnikiem platynek
	eLidFeederState									: E_Station; 							// Stan pracy podajnika platynek			
	eLidFeederRunningState							: E_LidFeederState; 					// Stan pracy podajnika platynek
	fbLidFeederState								: FB_State; 

	//Podajnik platynek 2
	fbLidFeeder2									: FB_LidFeeder; 						// Blok sterowania podajnikiem platynek
	eLidFeeder2State								: E_Station; 							// Stan pracy podajnika platynek			
	eLidFeeder2RunningState							: E_LidFeederState; 					// Stan pracy podajnika platynek
	fbLidFeeder2State								: FB_State; 

	QbLidFeederBlockActuator 				AT %Q*	: BOOL;  		// Blokada 
	
	// WEJŚCIA I WYJŚCIA SPRZĘTOWE 1
	QbLidFeeder_FeederActuator1						: BOOL; 				(*Pneu*) 		// Sterowanie zaworem podajnika platynek na wyspie zaworowej
	QbLidFeeder_FeederActuator2						: BOOL; 				(*Pneu*) 		// Sterowanie zaworem podajnika platynek na wyspie zaworowej
	QbLidFeeder_HeaterActuator						: BOOL;  				(*Pneu*) 		// Sterowanie zaworem grzałki platynek na wyspie zaworowej
	QbLidFeeder_SuckerActuator 				AT %Q*	: BOOL; 								// Sterowanie zaworem ssawki platynek na wyspie zaworowej
	QbLidFeederHeaterPWMOut 				AT %Q*	: BOOL; 								// Wyjście sterujące grzałką podajnika platynek
	

	AIbLidFeederHeaterTempCVSensor 			AT %I*	: INT; 									// Wartość aktualnej temperatury grzałki podajnika platynek
	IbLidFeederTempSensorFailure 			AT %I*	: BOOL; 								// Informacja o uszkodzeniu czujnika temperatury grzałki podajnika platynek
	QbLidFeeder_HeightMotorUp 				AT %Q*	: BOOL;									// Sterowanie silnikiem podnosnika stacji w górę 
	QbLidFeeder_HeightMotorDown 			AT %Q*	: BOOL;									//Sterowanie silnikiem podnosnika stacji w dół
	IbLidFeederHeightEncoderPulse  			AT %I* 	: BOOL;									// Wejście impulsów enkodera podnośnika platynek regulacji wysokości 
									// Czujnik niskiego pozimu platynek	
	
	// WEJŚCIA I WYJŚCIA SPRZĘTOWE 2		
	QbLidFeeder2_FeederActuator1					: BOOL; 				(*Pneu*) 		// Sterowanie zaworem podajnika platynek na wyspie zaworowej
	QbLidFeeder2_FeederActuator2					: BOOL; 				(*Pneu*) 		// Sterowanie zaworem podajnika platynek na wyspie zaworowej
	QbLidFeeder2_HeaterActuator						: BOOL;  				(*Pneu*) 		// Sterowanie zaworem grzałki platynek na wyspie zaworowej
	QbLidFeeder2_SuckerActuator 			AT %Q*	: BOOL; 								// Sterowanie zaworem ssawki platynek na wyspie zaworowej
	QbLidFeeder2HeaterPWMOut 				AT %Q*	: BOOL; 								// Wyjście sterujące grzałką podajnika platynek
	IbLidFeeder2UpSensor1 					AT %I*	: BOOL; 								// Czujnik pozycji górnej ssawki podajnika platynek
	IbLidFeeder2DownSensor1 				AT %I*	: BOOL;								
	IbLidFeeder2DownSensor2 				AT %I*	: BOOL;								
									// Czujnik zassania platynki
	AIbLidFeeder2HeaterTempCVSensor 		AT %I*	: INT; 									// Wartość aktualnej temperatury grzałki podajnika platynek
	IbLidFeeder2TempSensorFailure 			AT %I*	: BOOL; 								// Informacja o uszkodzeniu czujnika temperatury grzałki podajnika platynek
										// Czujnik niskiego pozimu platynek
	
	//Vasyl 24.10.25 Aktualizacja enkodera
	IbLidFeederHeightEncoderSetCDone		AT %I*: BOOL;	
	IudiLidFeederHeightEncoderCV         	AT %I*: UDINT; 	
	QbLidFeederHeightEncoderSetC 			AT %Q*: BOOL;		
	QudiLidFeederHeightEncoderSetCV       	AT %Q*: UDINT; 	
	
	tofLidFeederEnable								: TOF;
	tonLidFeederEnable								: TON;
	rtEnable										: R_TRIG;

	tonLidFeederCatchSensorClosed					: TON;
                	
	bTemp											: BOOL;
	bSimulation										: BOOL;
	
	bLidFeederWarning1								: BOOL;
	bLidFeederWarning2								: BOOL;
	
	//PRZECIAGANIE
	eLidFeederDragStation							: E_Station;
	eLidFeederDragRunningStation					: E_DragStationState;
	fbLidFeederDragState							: FB_State;
	fbLidFeederDragStation							: FB_FormsDragStepper;

	tofLidFeederDragStationEnable					: TOF;	
	
	//WEJSCIA I WYJSCIA SPRZETOWE
	QbLidFeederDragLeadBefore1Actuator        		: BOOL;				// Siłownikiem prowadzenia przed 1(1 faza)
	QbLidFeederDragLeadBefore2Actuator        		: BOOL;				// Siłownikiem prowadzenia przed 1(1 faza)
	
	
	IbLidFeederDragLeadBefore2UpSensor 				AT %I*  : BOOL;				// Czujnik
	
	bLidFeederUp									: BOOL;				//Podnoszenie podajników do góry
	
	
	//Chwytak formatek
	fbLidFeederFormPositioning						: FB_Gate;				// Bloczek obsługi bandy
	IbLidFeederFormPositioningUpSensor				AT %I*	: BOOL; 		// 
	QbLidFeederFormPositioningActuator 				: BOOL;  		



	
	bTestManual: BOOL;
END_VAR

//QbLidFeederBlockActuator	:= (GVL.eLidFeederPackageState[1].bFormPresent AND GVL.bFormTransportersDispencerCmdStart) OR 
//							   (GVL.eLidFeederPackageState[2].bFormPresent AND GVL.bFormTransportersDispencerCmdStart);

IF P00_PackML.fbPMLModeManager.eModeStatus = Tc3_PackML.E_PMLUnitMode.ePMLUnitMode_AUTOMATIC AND tofLidFeederEnable.Q THEN
	
	QbLidFeederBlockActuator :=	P00_PackML.fbPMLAuto.ePMLState = Tc3_PackML.E_PMLState.ePMLState_EXECUTE OR 
								P00_PackML.fbPMLAuto.ePMLState = Tc3_PackML.E_PMLState.ePMLState_STOPPING OR 
								P00_PackML.fbPMLAuto.ePMLState = Tc3_PackML.E_PMLState.ePMLState_STARTING;
								
ELSIF P00_PackML.fbPMLModeManager.eModeStatus = Tc3_PackML.E_PMLUnitMode.ePMLUnitMode_MANUAL THEN
	
	QbLidFeederBlockActuator	:= P06_LidSealer.fbLidSealer.bBlockActuator OR P06_LidSealer.fbLidSealer2.bBlockActuator OR VIS.bLidFeeder1ManualHeaterAct OR VIS.bLidFeeder2ManualHeaterAct OR
			VIS.bLidFeeder1Run OR VIS.bLidFeeder2Run OR VIS.bLidFeederEnableShow;
	
END_IF

bLidFeederUp	:= GVL_IO.IbEmergencyStopButton0Pressed OR GVL_IO.IbEmergencyStopButton1Pressed OR GVL_IO.IbEmergencyStopButton2Pressed OR {warning 'PI odkomentować'}
				   GVL_IO.IbEmergencyStopButton3Pressed OR GVL_IO.IbEmergencyStopButton4Pressed OR IbTurnTableEmergencyStopButtonPressed OR (*IbPucksInserterEmergencyStopButton0Pressed OR*) IbPucksInserterEmergencyStopButton1Pressed
				   OR P07_ROPP.IbROPPEmergencyStopButton0Pressed OR P07_ROPP.IbROPPEmergencyStopButton1Pressed 
				AND (QbLidFeeder_HeaterActuator OR QbLidFeeder2_HeaterActuator);
							   
ACT_LidFeeder();
ACT_LidFeeder2();
ACT_LidFeederDragStation();
a_LidFeederFormPositioning();
aLidFeederWarnings();

//GENEROWANIE STANU STACJI DO WIZKI
fbLidFeederState(
	eState 					:= eLidFeederState , 
	bRun 					:= VIS.bLidFeeder1PrepareRun OR VIS.bLidFeeder1Run,	
	eLidFeederRunningState 	:= eLidFeederRunningState , 
	sStateDesc				=> VIS.sLidFeeder1State,
	iState					=> VIS.iLidFeeder1State	);
	
fbLidFeeder2State(
	eState 					:= eLidFeeder2State , 
	bRun 					:= VIS.bLidFeeder2PrepareRun OR VIS.bLidFeeder2Run,	
	eLidFeederRunningState 	:= eLidFeeder2RunningState , 
	sStateDesc				=> VIS.sLidFeeder2State,
	iState					=> VIS.iLidFeeder2State	);
	
(* BAZOWANIE - ZMIAN*)
tonLidFeederEnable(IN := fbLidFeeder.bEnable, PT := T#2S); (*Dodany ton bo Wizka zjebnie wgrywa zmienne, najpierw włacza Enabla a potem dopiero wybiera recepture*)
rtEnable(CLK := tonLidFeederEnable.Q, Q=>);
IF rtEnable.Q AND (P00_PackML.fbPMLAuto.ePMLState = Tc3_PackML.E_PMLState.ePMLState_IDLE OR 
   P00_PackML.fbPMLAuto.ePMLState = Tc3_PackML.E_PMLState.ePMLState_EXECUTE) THEN
    VIS.bLidFeederHeightSet 		:= TRUE;
ELSIF (fbLidFeeder.eState = E_Station.eHomingDone AND fbLidFeeder2.eState = E_Station.eHomingDone)OR VIS.bErrorOccure THEN
    VIS.bLidFeederHeightSet 		:= FALSE;
END_IF
(*KONIEC BAZOWANIE - ZMIANA*)

//PRZEPISYWANIE POMIARÓW
VIS.lrLidFeeder1HeaterTempCV	:= (INT_TO_LREAL(AIbLidFeederHeaterTempCVSensor)/10);
VIS.lrLidFeeder2HeaterTempCV	:= (INT_TO_LREAL(AIbLidFeeder2HeaterTempCVSensor)/10);

//SYMULACJA CZUJNIKÓW IGLIC

//Opoznienie wyłączanie enabla
tofLidFeederEnable(IN:= VIS.bLidFeederEnableShow, PT:=T#2S);

//KASOWANIE ROZKAZÓW CYKLI
IF fbLidFeeder.bCycleDone AND GVL.bManualMode THEN
	VIS.bLidFeeder1PrepareRun 		:= FALSE;
	VIS.bLidFeeder1Run 			:= FALSE;
END_IF
IF fbLidFeeder2.bCycleDone AND GVL.bManualMode THEN
	VIS.bLidFeeder2PrepareRun 		:= FALSE;
	VIS.bLidFeeder2Run 			:= FALSE;
END_IF

IF bSimulation THEN
	IF fbLidFeeder.eState = E_Station.eReady AND fbLidFeeder2.eState = E_Station.eReady THEN
		VIS.bLidFeeder1PrepareRun	:= TRUE;
		VIS.bLidFeeder2PrepareRun	:= TRUE;
	END_IF
	IF fbLidFeeder.eState = E_Station.eRunning AND fbLidFeeder2.eState = E_Station.eRunning THEN
		
		IF (VIS.bLidFeeder1PrepareRun AND NOT VIS.bLidFeeder1Run AND IbLidFeederDownSensor1) AND
		   (VIS.bLidFeeder2PrepareRun AND NOT VIS.bLidFeeder2Run AND IbLidFeeder2DownSensor1) THEN		
			VIS.bLidFeeder1Run 	:= TRUE;
			VIS.bLidFeeder2Run 	:= TRUE;		
	
		END_IF
	END_IF
	
	IF fbLidFeeder.bCycleDone AND fbLidFeeder2.bCycleDone THEN
		
		VIS.bLidFeeder1PrepareRun	:= FALSE;
		VIS.bLidFeeder2PrepareRun	:= FALSE;
		VIS.bLidFeeder1Run 		:= FALSE;
		VIS.bLidFeeder2Run 		:= FALSE;
		
	END_IF
END_IF

(*
{warning: 'Sprawdzic działanie czujnika niskiego poziomu - kiedy stan wysoki'}

//Ostrzeżenia Podajnik 1 
GVL.LidFeederWarning[0].sDescription			:= 'Niski poziom platynek podajnik 1';

IF bLidFeederWarning1 AND NOT GVL.LidFeederWarning[0].bWarning THEN
	
	GVL.LidFeederWarning[0].bWarning			:= TRUE;
	
ELSIF NOT bLidFeederWarning1 AND GVL.LidFeederWarning[0].bAcknowledge THEN
	
	GVL.LidFeederWarning[0].bWarning			:= FALSE;
	GVL.LidFeederWarning[0].bAcknowledge		:= FALSE;
	//GvlVisualization.uliWarningAcknowledge.4 	:= FALSE;
	
ELSIF GVL.LidFeederWarning[0].bAcknowledge THEN
{warning: 'Sprawdzic potwierdzenie warningu tutaj i wewnatrz bloczka gdy zmieni sie stan czujnika '}	
	bLidFeederWarning1							:= FALSE;
	GVL.LidFeederWarning[0].bAcknowledge		:= TRUE;
	
END_IF

//Ostrzeżenia Podajnik 2 
GVL.LidFeederWarning[1].sDescription			:= 'Niski poziom platynek podajnik 2';

IF bLidFeederWarning2 AND NOT GVL.LidFeederWarning[1].bWarning THEN
	
	GVL.LidFeederWarning[1].bWarning			:= TRUE;
	
ELSIF NOT bLidFeederWarning2 AND GVL.LidFeederWarning[1].bAcknowledge THEN
	
	GVL.LidFeederWarning[1].bWarning			:= FALSE;
	GVL.LidFeederWarning[1].bAcknowledge		:= FALSE;
	//GvlVisualization.uliWarningAcknowledge.4 	:= FALSE;
	
ELSIF GVL.LidFeederWarning[1].bAcknowledge THEN
	
	bLidFeederWarning2							:= FALSE;	
	GVL.LidFeederWarning[1].bAcknowledge		:= TRUE;
	
END_IF
*)

//Przeciąganie
tofLidFeederDragStationEnable(IN:= VIS.bLidFeederDragingStationEnableShow, PT:= T#2S);

ACTION a_LidFeederFormPositioning:
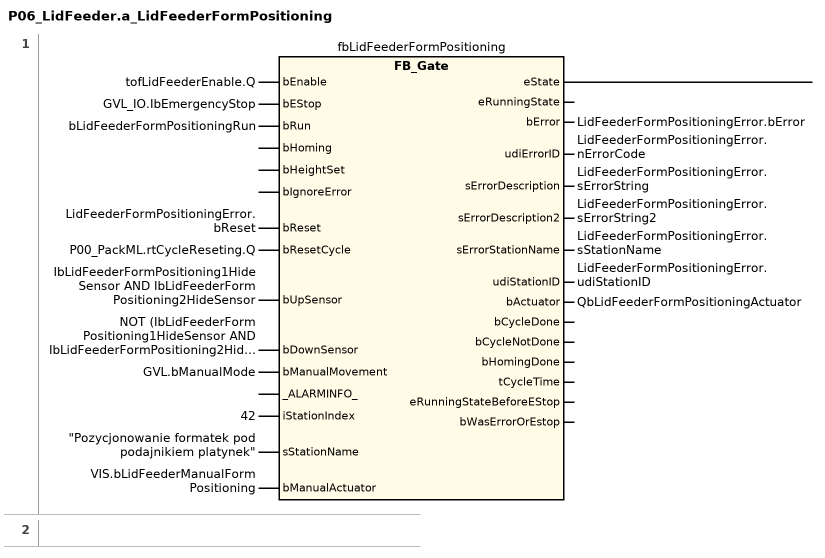
// NETWORK 1
fbLidFeederFormPositioning(
    bEnable := tofLidFeederEnable.Q,
    bEStop := GVL_IO.IbEmergencyStop,
    bRun := bLidFeederFormPositioningRun,
    bReset := LidFeederFormPositioningError.bReset,
    bResetCycle := P00_PackML.rtCycleReseting.Q,
    bUpSensor := IbLidFeederFormPositioning1HideSensor AND IbLidFeederFormPositioning2HideSensor,
    bDownSensor := NOT (IbLidFeederFormPositioning1HideSensor AND IbLidFeederFormPositioning2HideSensor),
    bManualMovement := GVL.bManualMode,
    iStationIndex := 42,
    sStationName := "Pozycjonowanie formatek pod podajnikiem platynek",
    bManualActuator := VIS.bLidFeederManualFormPositioning,
    bError => LidFeederFormPositioningError.bError,
    udiErrorID => LidFeederFormPositioningError.nErrorCode,
    sErrorDescription => LidFeederFormPositioningError.sErrorString,
    sErrorDescription2 => LidFeederFormPositioningError.sErrorString2,
    sErrorStationName => LidFeederFormPositioningError.sStationName,
    udiStationID => LidFeederFormPositioningError.udiStationID,
    bActuator => QbLidFeederFormPositioningActuator); // FB_Gate

// NETWORK 2
END_ACTION

ACTION ACT_LidFeeder:
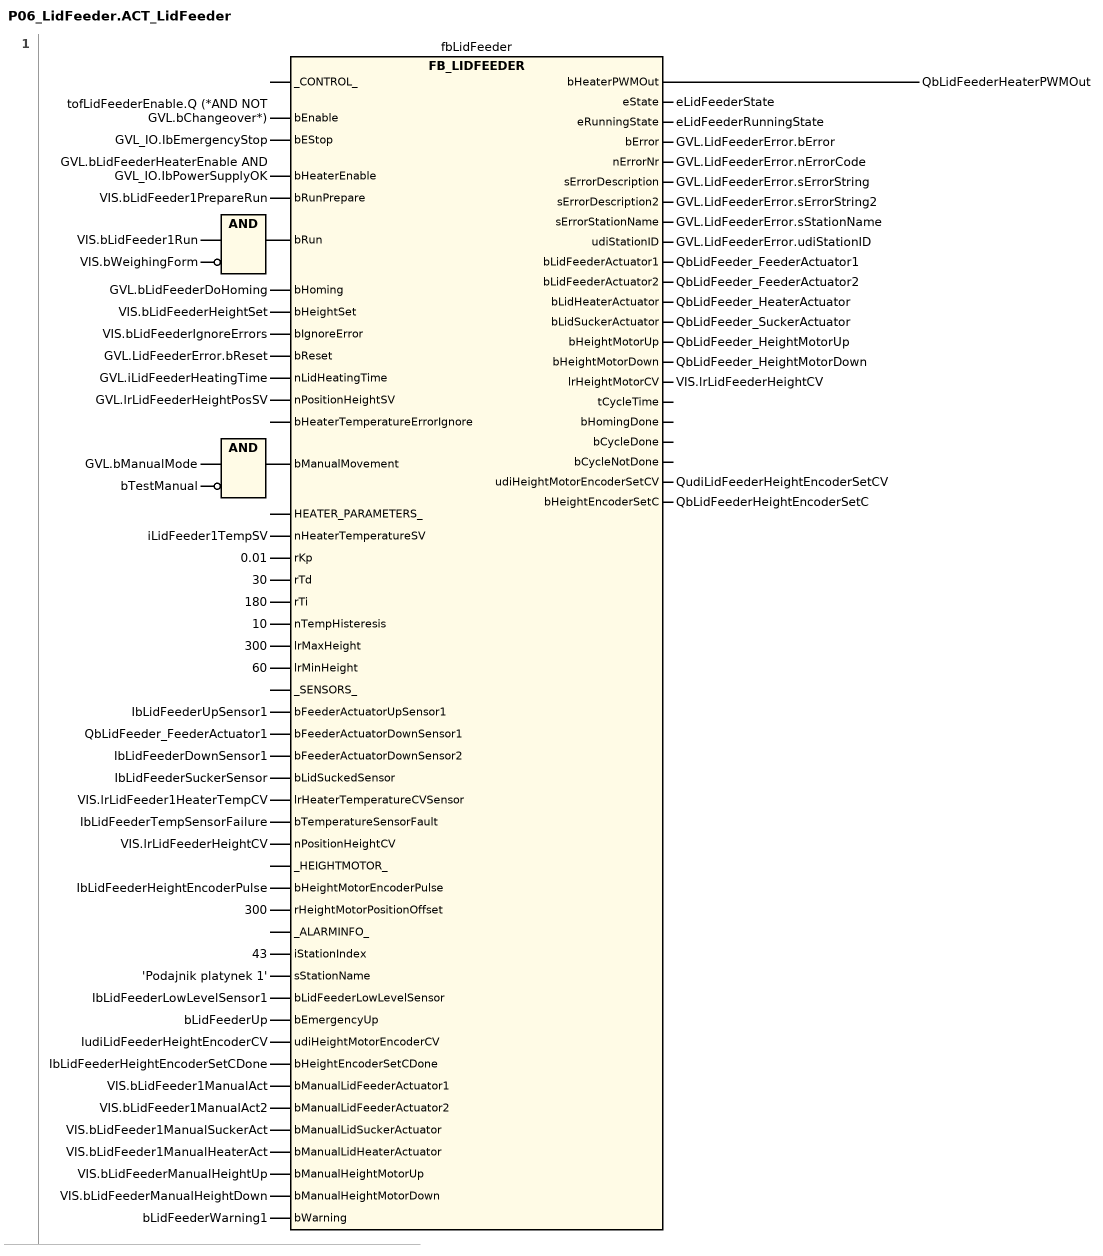
// NETWORK 1
fbLidFeeder(
    bEnable := tofLidFeederEnable.Q (*AND NOT GVL.bChangeover*),
    bEStop := GVL_IO.IbEmergencyStop,
    bHeaterEnable := GVL.bLidFeederHeaterEnable AND GVL_IO.IbPowerSupplyOK,
    bRunPrepare := VIS.bLidFeeder1PrepareRun,
    bRun := VIS.bLidFeeder1Run AND NOT VIS.bWeighingForm,
    bHoming := GVL.bLidFeederDoHoming,
    bHeightSet := VIS.bLidFeederHeightSet,
    bIgnoreError := VIS.bLidFeederIgnoreErrors,
    bReset := GVL.LidFeederError.bReset,
    nLidHeatingTime := GVL.iLidFeederHeatingTime,
    nPositionHeightSV := GVL.lrLidFeederHeightPosSV,
    bManualMovement := GVL.bManualMode AND NOT bTestManual,
    nHeaterTemperatureSV := iLidFeeder1TempSV,
    rKp := 0.01,
    rTd := 30,
    rTi := 180,
    nTempHisteresis := 10,
    lrMaxHeight := 300,
    lrMinHeight := 60,
    bFeederActuatorUpSensor1 := IbLidFeederUpSensor1,
    bFeederActuatorDownSensor1 := QbLidFeeder_FeederActuator1,
    bFeederActuatorDownSensor2 := IbLidFeederDownSensor1,
    bLidSuckedSensor := IbLidFeederSuckerSensor,
    lrHeaterTemperatureCVSensor := VIS.lrLidFeeder1HeaterTempCV,
    bTemperatureSensorFault := IbLidFeederTempSensorFailure,
    nPositionHeightCV := VIS.lrLidFeederHeightCV,
    bHeightMotorEncoderPulse := IbLidFeederHeightEncoderPulse,
    rHeightMotorPositionOffset := 300,
    iStationIndex := 43,
    sStationName := 'Podajnik platynek 1',
    bLidFeederLowLevelSensor := IbLidFeederLowLevelSensor1,
    bEmergencyUp := bLidFeederUp,
    udiHeightMotorEncoderCV := IudiLidFeederHeightEncoderCV,
    bHeightEncoderSetCDone := IbLidFeederHeightEncoderSetCDone,
    bManualLidFeederActuator1 := VIS.bLidFeeder1ManualAct,
    bManualLidFeederActuator2 := VIS.bLidFeeder1ManualAct2,
    bManualLidSuckerActuator := VIS.bLidFeeder1ManualSuckerAct,
    bManualLidHeaterActuator := VIS.bLidFeeder1ManualHeaterAct,
    bManualHeightMotorUp := VIS.bLidFeederManualHeightUp,
    bManualHeightMotorDown := VIS.bLidFeederManualHeightDown,
    bWarning := bLidFeederWarning1,
    eState => eLidFeederState,
    eRunningState => eLidFeederRunningState,
    bError => GVL.LidFeederError.bError,
    nErrorNr => GVL.LidFeederError.nErrorCode,
    sErrorDescription => GVL.LidFeederError.sErrorString,
    sErrorDescription2 => GVL.LidFeederError.sErrorString2,
    sErrorStationName => GVL.LidFeederError.sStationName,
    udiStationID => GVL.LidFeederError.udiStationID,
    bLidFeederActuator1 => QbLidFeeder_FeederActuator1,
    bLidFeederActuator2 => QbLidFeeder_FeederActuator2,
    bLidHeaterActuator => QbLidFeeder_HeaterActuator,
    bLidSuckerActuator => QbLidFeeder_SuckerActuator,
    bHeightMotorUp => QbLidFeeder_HeightMotorUp,
    bHeightMotorDown => QbLidFeeder_HeightMotorDown,
    lrHeightMotorCV => VIS.lrLidFeederHeightCV,
    udiHeightMotorEncoderSetCV => QudiLidFeederHeightEncoderSetCV,
    bHeightEncoderSetC => QbLidFeederHeightEncoderSetC); // FB_LIDFEEDER
QbLidFeederHeaterPWMOut := fbLidFeeder.bHeaterPWMOut;
END_ACTION

ACTION ACT_LidFeeder2:
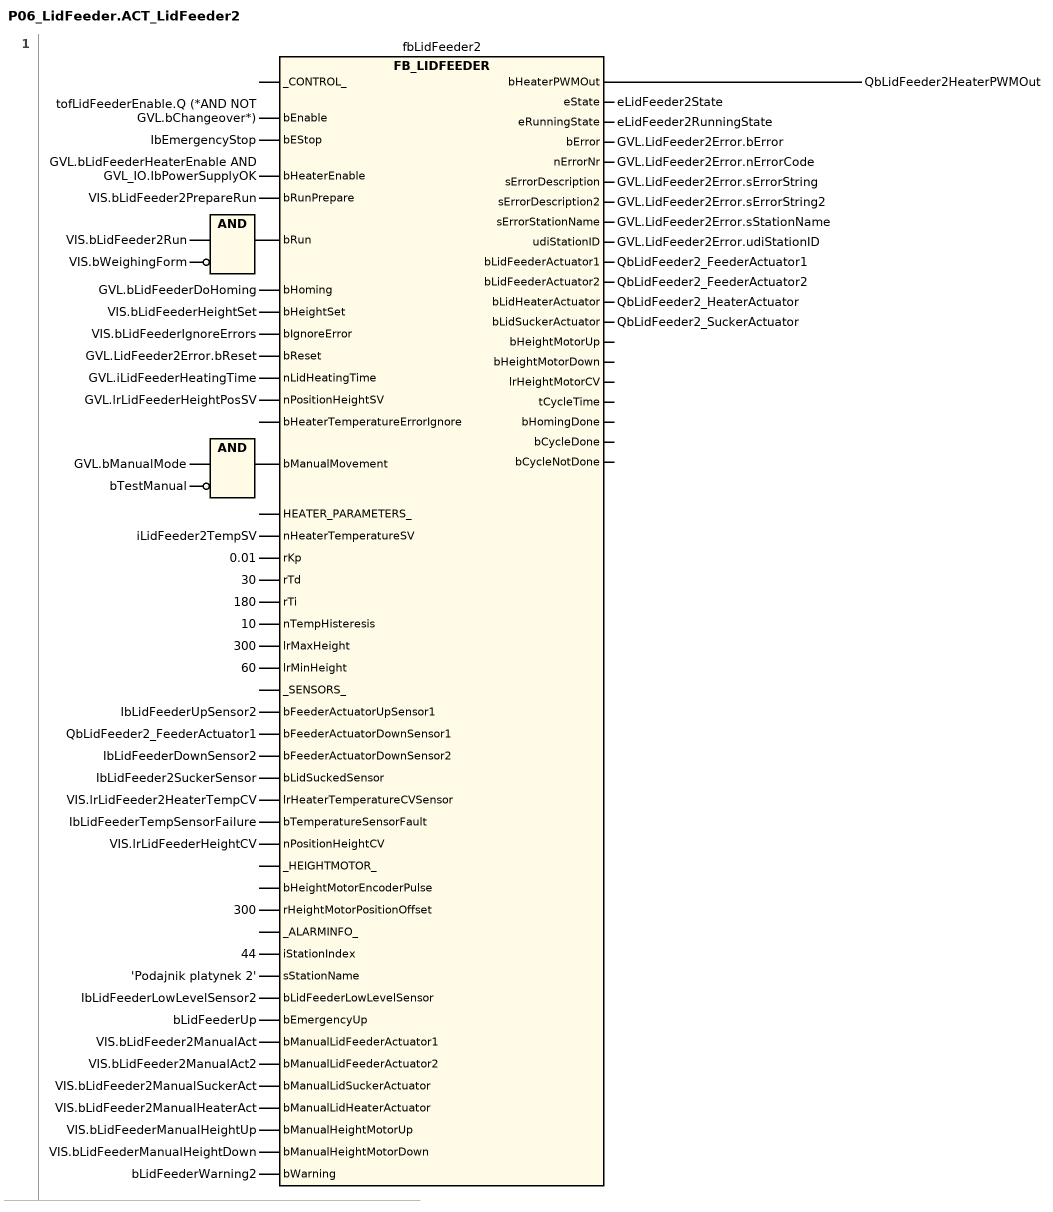
// NETWORK 1
fbLidFeeder2(
    bEnable := tofLidFeederEnable.Q (*AND NOT GVL.bChangeover*),
    bEStop := IbEmergencyStop,
    bHeaterEnable := GVL.bLidFeederHeaterEnable AND GVL_IO.IbPowerSupplyOK,
    bRunPrepare := VIS.bLidFeeder2PrepareRun,
    bRun := VIS.bLidFeeder2Run AND NOT VIS.bWeighingForm,
    bHoming := GVL.bLidFeederDoHoming,
    bHeightSet := VIS.bLidFeederHeightSet,
    bIgnoreError := VIS.bLidFeederIgnoreErrors,
    bReset := GVL.LidFeeder2Error.bReset,
    nLidHeatingTime := GVL.iLidFeederHeatingTime,
    nPositionHeightSV := GVL.lrLidFeederHeightPosSV,
    bManualMovement := GVL.bManualMode AND NOT bTestManual,
    nHeaterTemperatureSV := iLidFeeder2TempSV,
    rKp := 0.01,
    rTd := 30,
    rTi := 180,
    nTempHisteresis := 10,
    lrMaxHeight := 300,
    lrMinHeight := 60,
    bFeederActuatorUpSensor1 := IbLidFeederUpSensor2,
    bFeederActuatorDownSensor1 := QbLidFeeder2_FeederActuator1,
    bFeederActuatorDownSensor2 := IbLidFeederDownSensor2,
    bLidSuckedSensor := IbLidFeeder2SuckerSensor,
    lrHeaterTemperatureCVSensor := VIS.lrLidFeeder2HeaterTempCV,
    bTemperatureSensorFault := IbLidFeederTempSensorFailure,
    nPositionHeightCV := VIS.lrLidFeederHeightCV,
    rHeightMotorPositionOffset := 300,
    iStationIndex := 44,
    sStationName := 'Podajnik platynek 2',
    bLidFeederLowLevelSensor := IbLidFeederLowLevelSensor2,
    bEmergencyUp := bLidFeederUp,
    bManualLidFeederActuator1 := VIS.bLidFeeder2ManualAct,
    bManualLidFeederActuator2 := VIS.bLidFeeder2ManualAct2,
    bManualLidSuckerActuator := VIS.bLidFeeder2ManualSuckerAct,
    bManualLidHeaterActuator := VIS.bLidFeeder2ManualHeaterAct,
    bManualHeightMotorUp := VIS.bLidFeederManualHeightUp,
    bManualHeightMotorDown := VIS.bLidFeederManualHeightDown,
    bWarning := bLidFeederWarning2,
    eState => eLidFeeder2State,
    eRunningState => eLidFeeder2RunningState,
    bError => GVL.LidFeeder2Error.bError,
    nErrorNr => GVL.LidFeeder2Error.nErrorCode,
    sErrorDescription => GVL.LidFeeder2Error.sErrorString,
    sErrorDescription2 => GVL.LidFeeder2Error.sErrorString2,
    sErrorStationName => GVL.LidFeeder2Error.sStationName,
    udiStationID => GVL.LidFeeder2Error.udiStationID,
    bLidFeederActuator1 => QbLidFeeder2_FeederActuator1,
    bLidFeederActuator2 => QbLidFeeder2_FeederActuator2,
    bLidHeaterActuator => QbLidFeeder2_HeaterActuator,
    bLidSuckerActuator => QbLidFeeder2_SuckerActuator); // FB_LIDFEEDER
QbLidFeeder2HeaterPWMOut := fbLidFeeder2.bHeaterPWMOut;
END_ACTION

ACTION ACT_LidFeederDragStation:
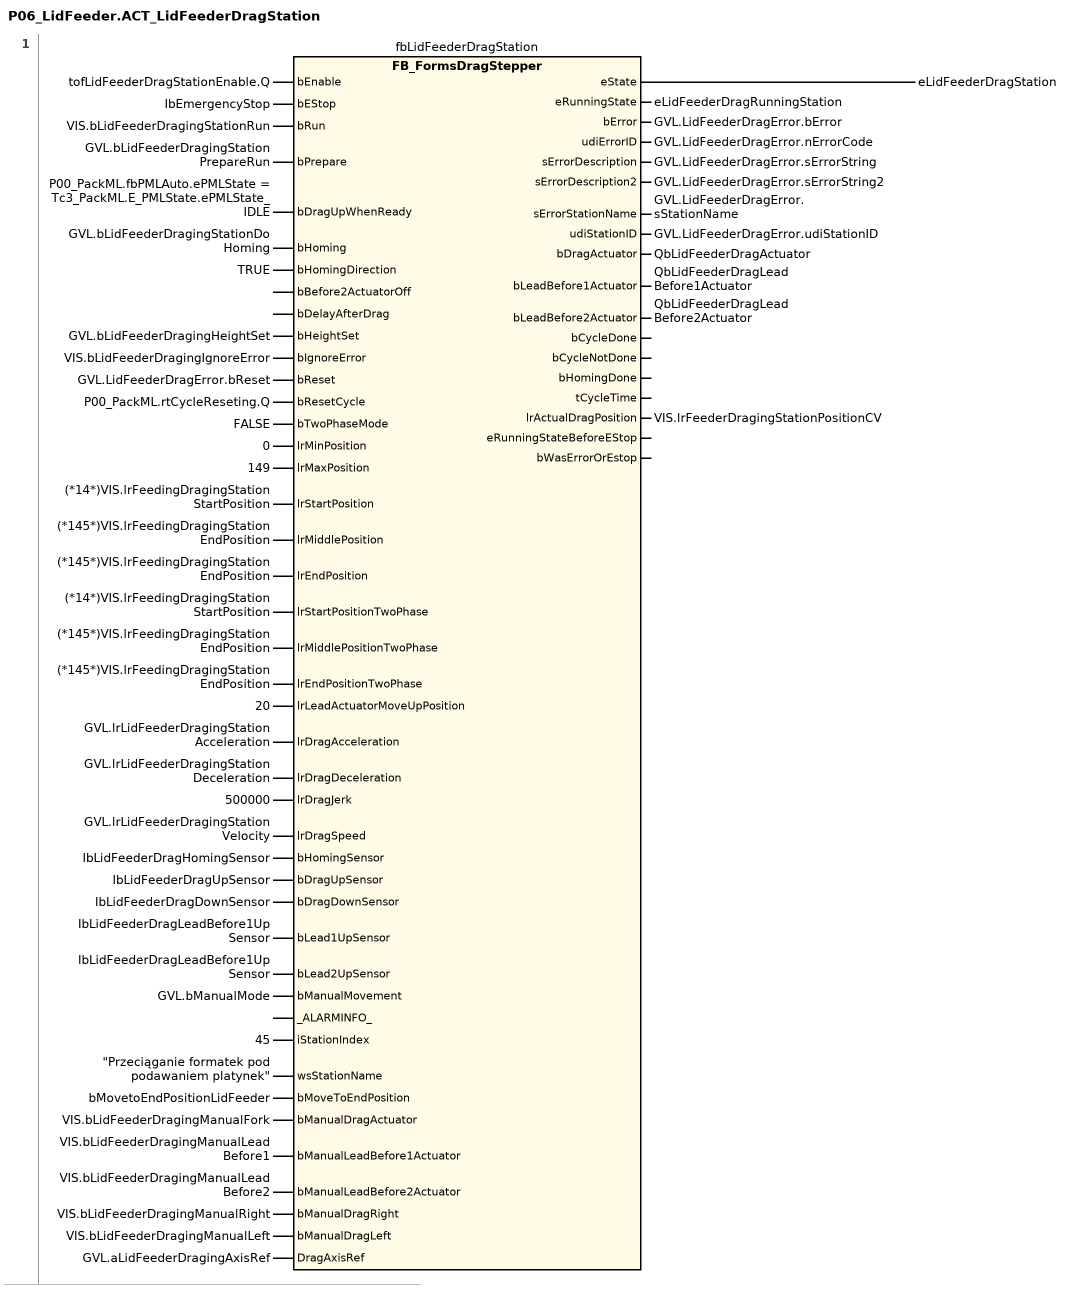
// NETWORK 1
fbLidFeederDragStation(
    bEnable := tofLidFeederDragStationEnable.Q,
    bEStop := IbEmergencyStop,
    bRun := VIS.bLidFeederDragingStationRun,
    bPrepare := GVL.bLidFeederDragingStationPrepareRun,
    bDragUpWhenReady := P00_PackML.fbPMLAuto.ePMLState = Tc3_PackML.E_PMLState.ePMLState_IDLE,
    bHoming := GVL.bLidFeederDragingStationDoHoming,
    bHomingDirection := TRUE,
    bHeightSet := GVL.bLidFeederDragingHeightSet,
    bIgnoreError := VIS.bLidFeederDragingIgnoreError,
    bReset := GVL.LidFeederDragError.bReset,
    bResetCycle := P00_PackML.rtCycleReseting.Q,
    bTwoPhaseMode := FALSE,
    lrMinPosition := 0,
    lrMaxPosition := 149,
    lrStartPosition := (*14*)VIS.lrFeedingDragingStationStartPosition,
    lrMiddlePosition := (*145*)VIS.lrFeedingDragingStationEndPosition,
    lrEndPosition := (*145*)VIS.lrFeedingDragingStationEndPosition,
    lrStartPositionTwoPhase := (*14*)VIS.lrFeedingDragingStationStartPosition,
    lrMiddlePositionTwoPhase := (*145*)VIS.lrFeedingDragingStationEndPosition,
    lrEndPositionTwoPhase := (*145*)VIS.lrFeedingDragingStationEndPosition,
    lrLeadActuatorMoveUpPosition := 20,
    lrDragAcceleration := GVL.lrLidFeederDragingStationAcceleration,
    lrDragDeceleration := GVL.lrLidFeederDragingStationDeceleration,
    lrDragJerk := 500000,
    lrDragSpeed := GVL.lrLidFeederDragingStationVelocity,
    bHomingSensor := IbLidFeederDragHomingSensor,
    bDragUpSensor := IbLidFeederDragUpSensor,
    bDragDownSensor := IbLidFeederDragDownSensor,
    bLead1UpSensor := IbLidFeederDragLeadBefore1UpSensor,
    bLead2UpSensor := IbLidFeederDragLeadBefore1UpSensor,
    bManualMovement := GVL.bManualMode,
    iStationIndex := 45,
    wsStationName := "Przeciąganie formatek pod podawaniem platynek",
    bMoveToEndPosition := bMovetoEndPositionLidFeeder,
    bManualDragActuator := VIS.bLidFeederDragingManualFork,
    bManualLeadBefore1Actuator := VIS.bLidFeederDragingManualLeadBefore1,
    bManualLeadBefore2Actuator := VIS.bLidFeederDragingManualLeadBefore2,
    bManualDragRight := VIS.bLidFeederDragingManualRight,
    bManualDragLeft := VIS.bLidFeederDragingManualLeft,
    DragAxisRef := GVL.aLidFeederDragingAxisRef,
    eRunningState => eLidFeederDragRunningStation,
    bError => GVL.LidFeederDragError.bError,
    udiErrorID => GVL.LidFeederDragError.nErrorCode,
    sErrorDescription => GVL.LidFeederDragError.sErrorString,
    sErrorDescription2 => GVL.LidFeederDragError.sErrorString2,
    sErrorStationName => GVL.LidFeederDragError.sStationName,
    udiStationID => GVL.LidFeederDragError.udiStationID,
    bDragActuator => QbLidFeederDragActuator,
    bLeadBefore1Actuator => QbLidFeederDragLeadBefore1Actuator,
    bLeadBefore2Actuator => QbLidFeederDragLeadBefore2Actuator,
    lrActualDragPosition => VIS.lrFeederDragingStationPositionCV); // FB_FormsDragStepper
eLidFeederDragStation := fbLidFeederDragStation.eState;
END_ACTION

ACTION ACT_Limits:
(*
Nazwa:			aSetRecipe
Opis:			Zapisywanie zmiennych gdy mają wartość 0 
Wersja:			v0.1
Data:			2022-06-22
Autor:			DP
Urzadzenia:		
Konfiguracja:	
Info:
- zabezpieczenie przed recepturami które nie mają tych parametrów i jest w nich wartość 0
*)

IF 	VIS.lrFeedingDragingStationStartPosition		= 0		THEN	VIS.lrFeedingDragingStationStartPosition		:=	14;		END_IF;
IF 	VIS.lrFeedingDragingStationEndPosition		= 0		THEN	VIS.lrFeedingDragingStationEndPosition		:=	145;	END_IF;
END_ACTION

ACTION aLidFeederWarnings:

//Warning 0
LidFeederWarning[0].sDescription:='Podajnik platynek 1 | Brak platynek w zasobniku';
IF bLidFeederWarning1 AND NOT LidFeederWarning[0].bWarning AND bLidFeederEnable THEN
	LidFeederWarning[0].bWarning:=TRUE;
ELSIF NOT bLidFeederWarning1 AND LidFeederWarning[0].bAcknowledge THEN
	LidFeederWarning[0].bWarning		:=	FALSE;
	LidFeederWarning[0].bAcknowledge	:=	FALSE;
	VIS.uliWarningOccure.39				:=	FALSE;
ELSIF LidFeederWarning[0].bAcknowledge THEN
	LidFeederWarning[0].bAcknowledge	:=	TRUE;
END_IF

//Warning 1
LidFeederWarning[1].sDescription:='Podajnik platynek 2 | Brak platynek w zasobniku';
IF bLidFeederWarning2 AND NOT LidFeederWarning[1].bWarning AND bLidFeederEnable THEN
	LidFeederWarning[1].bWarning:=TRUE;
ELSIF NOT bLidFeederWarning2 AND LidFeederWarning[1].bAcknowledge THEN
	LidFeederWarning[1].bWarning		:=	FALSE;
	LidFeederWarning[1].bAcknowledge	:=	FALSE;
	VIS.uliWarningOccure.40				:=	FALSE;
ELSIF LidFeederWarning[1].bAcknowledge THEN
	LidFeederWarning[1].bAcknowledge	:=	TRUE;
END_IF
END_ACTION

END_PROGRAM

// ---- POUs/FB/FB_LidFeeder.TcPOU
(*
Nazwa:			FB_LidFeeder
Opis:			Podajnik platynek
Wersja:			v1.1
Data:			2024-08-28
Autor:			TW,DP,MP
Urzadzenia:		Podnosnik stacji, grzałka, czujnik temp, ssawka
Konfiguracja:	
Info: 
- [20240918] [DP] Estop De
- [20240828] [DP] poprawa control done
- dodany drugi siłownik
- dodano błędy od nastaw powyżej max i min (error 7 i 8)
- zmiana 11 wychodzenie z HeaterNotReady jak Homing
- Dodano HomingNeeded
- Zmiana Homingów według CatchStation
*)


